KUKA KRL program: FrED_Main.src, FrED_Main.dat

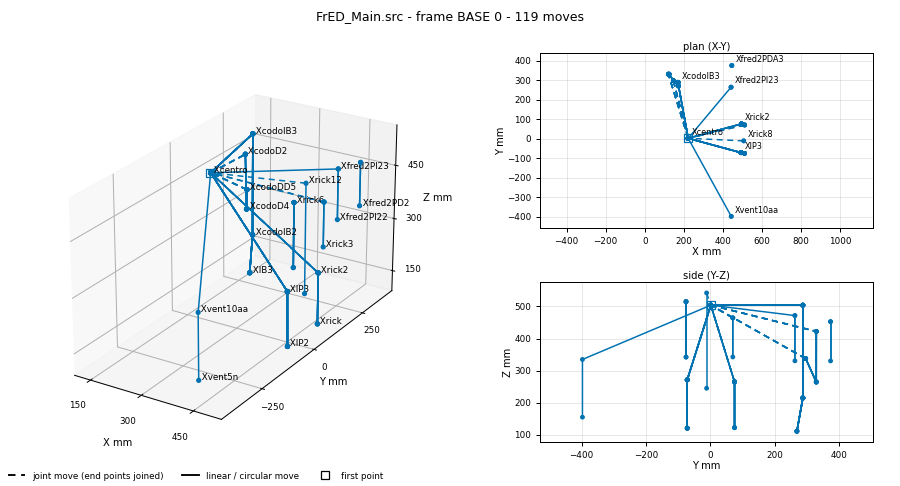
[picture p0: tool path of FrED_Main.src in frame BASE 0, 119 of 201 moves have a stored position in this frame; points joined in program order, loops and branches not executed]
--- FrED_Main.src ---
&ACCESS RVO
&PARAM DISKPATH = KRC:\R1\AAWS3
DEF codigoWS3( )
;FOLD INI;%{PE}
   DECL INT i
  ;FOLD BASISTECH INI
    GLOBAL INTERRUPT DECL 3 WHEN $STOPMESS==TRUE DO IR_STOPM ( )
    INTERRUPT ON 3
    BAS (#INITMOV,0 )

  ;ENDFOLD (BASISTECH INI)
;FOLD SPOTTECH INIw
USERSPOT(#INIT)
;ENDFOLD (SPOTTECH INI)
;FOLD GRIPPERTECH INI
USER_GRP(0,DUMMY,DUMMY,GDEFAULT)
;ENDFOLD (GRIPPERTECH INI)
;FOLD USER INI
  ;Make your modifications here
;ENDFOLD (USER INI)

;ENDFOLD (INI)

INTERRUPT DECL 25 WHEN NOT $IN[107] DO PAUSA()


;FOLD WAIT FOR ( IN 107 '' );%{PE}%R 8.3.40,%MKUKATPBASIS,%CEXT_WAIT_FOR,%VEXT_WAIT_FOR,%P 2:, 4:, 5:$IN, 6:107, 7:, 9:
WAIT FOR  ( $IN[107] )
;ENDFOLD
$OUT[105]=TRUE

INTERRUPT ON 25

FOR i= 1 to 2 STEP +1


;---------------------------------------------------------------------------------------------------------------------------------------------------------
;FRED 1


$OUT[101] = FALSE
WAIT SEC 0.5

;FOLD ; hola;%{PE}%R 8.3.40,%MKUKATPBASIS,%CCOMMENT,%VNORMAL,%P 2:hola
;ENDFOLD
;--- Movimiento a centro con velocidad reducida ---
PDAT_ACT=PPDAT4
FDAT_ACT=Fcentro
BAS(#PTP_PARAMS,20)
PTP Xcentro

;--- Abrir gripper ---
$OUT[101] = TRUE
$OUT[102] = FALSE
WAIT SEC 1

;--- Movimiento a codoIB3 ---
LDAT_ACT=LCPDAT2
FDAT_ACT=FcodoIB3
BAS(#CP_PARAMS,10)
LIN XcodoIB3

;--- Movimiento a codoIB2 ---
LDAT_ACT=LCPDAT5
FDAT_ACT=FcodoIB2
BAS(#CP_PARAMS,10)
LIN XcodoIB2

;FOLD LIN IB3 Vel=2 m/s CPDAT45 Tool[1]:navaja Base[0];%{PE}%R 8.3.40,%MKUKATPBASIS,%CMOVE,%VLIN,%P 1:LIN, 2:IB3, 3:, 5:2, 7:CPDAT45
$BWDSTART=FALSE
LDAT_ACT=LCPDAT45
FDAT_ACT=FIB3
BAS(#CP_PARAMS,2)
LIN XIB3
;ENDFOLD

;--- Cerrar gripper ---
$OUT[101] = FALSE
$OUT[102] = TRUE
WAIT SEC 1

;--- Regreso por codoIB2 ---
LDAT_ACT=LCPDAT5
FDAT_ACT=FcodoIB2
BAS(#CP_PARAMS,10)
LIN XcodoIB2

;--- Regreso por codoIB3 ---
LDAT_ACT=LCPDAT2
FDAT_ACT=FcodoIB3
BAS(#CP_PARAMS,10)
LIN XcodoIB3

;--- Regreso a centro ---
PDAT_ACT=PPDAT4
FDAT_ACT=Fcentro
BAS(#PTP_PARAMS,20)
PTP Xcentro

;FOLD LIN IP3 Vel=2 m/s CPDAT47 Tool[1]:navaja Base[0];%{PE}%R 8.3.40,%MKUKATPBASIS,%CMOVE,%VLIN,%P 1:LIN, 2:IP3, 3:, 5:2, 7:CPDAT47
$BWDSTART=FALSE
LDAT_ACT=LCPDAT47
FDAT_ACT=FIP3
BAS(#CP_PARAMS,2)
LIN XIP3
;ENDFOLD

;FOLD LIN IP2 Vel=2 m/s CPDAT46 Tool[1]:navaja Base[0];%{PE}%R 8.3.40,%MKUKATPBASIS,%CMOVE,%VLIN,%P 1:LIN, 2:IP2, 3:, 5:2, 7:CPDAT46
$BWDSTART=FALSE
LDAT_ACT=LCPDAT46
FDAT_ACT=FIP2
BAS(#CP_PARAMS,0.1)
LIN XIP2
;ENDFOLD


;--- Abrir gripper ---
$OUT[101] = TRUE
$OUT[102] = FALSE
WAIT SEC 1

;FOLD LIN IP4 Vel=2 m/s CPDAT47 Tool[1]:navaja Base[0];%{PE}%R 8.3.40,%MKUKATPBASIS,%CMOVE,%VLIN,%P 1:LIN, 2:IP4, 3:, 5:2, 7:CPDAT47
$BWDSTART=FALSE
LDAT_ACT=LCPDAT60
FDAT_ACT=FIP4
BAS(#CP_PARAMS,0.1)
LIN XIP4
;ENDFOLD



;--- Movimiento a centro ---
PDAT_ACT=PPDAT4
FDAT_ACT=Fcentro
BAS(#PTP_PARAMS,20)
PTP Xcentro

;--- Movimiento a codoD2 ---
PDAT_ACT=PPDAT6
FDAT_ACT=FcodoD2
BAS(#PTP_PARAMS,20)
PTP XcodoD2

;FOLD ; codoDnuevoagsrrar;%{PE}%R 8.3.40,%MKUKATPBASIS,%CCOMMENT,%VNORMAL,%P 2:codoDnuevoagsrrar
;ENDFOLD
;FOLD LIN codoD4 Vel=2 m/s CPDAT66 Tool[1]:navaja Base[0];%{PE}%R 8.3.40,%MKUKATPBASIS,%CMOVE,%VLIN,%P 1:LIN, 2:codoD4, 3:, 5:2, 7:CPDAT66
$BWDSTART=FALSE
LDAT_ACT=LCPDAT66
FDAT_ACT=FcodoD4
BAS(#CP_PARAMS,2)
LIN XcodoD4
;ENDFOLD

;--- Cerrar gripper ---
$OUT[101] = FALSE
$OUT[102] = TRUE
WAIT SEC 1

;FOLD LIN codoDD5 Vel=2 m/s CPDAT68 Tool[1]:navaja Base[0];%{PE}%R 8.3.40,%MKUKATPBASIS,%CMOVE,%VLIN,%P 1:LIN, 2:codoDD5, 3:, 5:2, 7:CPDAT68
$BWDSTART=FALSE
LDAT_ACT=LCPDAT68
FDAT_ACT=FcodoDD5
BAS(#CP_PARAMS,2)
LIN XcodoDD5
;ENDFOLD

;--- Movimiento a centro_5 con velocidad reducida ---
PDAT_ACT=PPDAT20
FDAT_ACT=Fcentro_5
BAS(#PTP_PARAMS,20)
PTP Xcentro_5

;FOLD LIN rick2 Vel=2 m/s CPDAT53 Tool[1]:navaja Base[0];%{PE}%R 8.3.40,%MKUKATPBASIS,%CMOVE,%VLIN,%P 1:LIN, 2:rick2, 3:, 5:2, 7:CPDAT53
$BWDSTART=FALSE
LDAT_ACT=LCPDAT53
FDAT_ACT=Frick2
BAS(#CP_PARAMS,2)
LIN Xrick2
;ENDFOLD

;FOLD LIN rick Vel=2 m/s CPDAT51 Tool[1]:navaja Base[0];%{PE}%R 8.3.40,%MKUKATPBASIS,%CMOVE,%VLIN,%P 1:LIN, 2:rick, 3:, 5:2, 7:CPDAT51
$BWDSTART=FALSE
LDAT_ACT=LCPDAT51
FDAT_ACT=Frick
BAS(#CP_PARAMS,0.1)
LIN Xrick
;ENDFOLD

;--- Abrir gripper ---
$OUT[101] = TRUE
$OUT[102] = FALSE
WAIT SEC 1

;FOLD LIN rick9 Vel=2 m/s CPDAT53 Tool[1]:navaja Base[0];%{PE}%R 8.3.40,%MKUKATPBASIS,%CMOVE,%VLIN,%P 1:LIN, 2:rick9, 3:, 5:2, 7:CPDAT53
$BWDSTART=FALSE
LDAT_ACT=LCPDAT61
FDAT_ACT=Frick9
BAS(#CP_PARAMS,0.1)
LIN Xrick9
;ENDFOLD

;--- Movimiento a centro ---
PDAT_ACT=PPDAT4
FDAT_ACT=Fcentro
BAS(#PTP_PARAMS,20)
PTP Xcentro

;FOLD LIN fred1PIA Vel=2 m/s CPDAT241 Tool[1]:navaja Base[0];%{PE}%R 8.3.40,%MKUKATPBASIS,%CMOVE,%VLIN,%P 1:LIN, 2:fred1PIA, 3:, 5:2, 7:CPDAT241
$BWDSTART=FALSE
LDAT_ACT=LCPDAT241
FDAT_ACT=Ffred1PIA
BAS(#CP_PARAMS,2)
LIN Xfred1PIA
;ENDFOLD

;FOLD LIN fred1PI Vel=2 m/s CPDAT240 Tool[1]:navaja Base[0];%{PE}%R 8.3.40,%MKUKATPBASIS,%CMOVE,%VLIN,%P 1:LIN, 2:fred1PI, 3:, 5:2, 7:CPDAT240
$BWDSTART=FALSE
LDAT_ACT=LCPDAT240
FDAT_ACT=Ffred1PI
BAS(#CP_PARAMS,2)
LIN Xfred1PI
;ENDFOLD

;--- Cerrar gripper ---
$OUT[101] = FALSE
$OUT[102] = TRUE
WAIT SEC 1

;FOLD LIN fred1PIA_1 Vel=2 m/s CPDAT241 Tool[1]:navaja Base[0];%{PE}%R 8.3.40,%MKUKATPBASIS,%CMOVE,%VLIN,%P 1:LIN, 2:fred1PIA_1, 3:, 5:2, 7:CPDAT241
$BWDSTART=FALSE
LDAT_ACT=LCPDAT244
FDAT_ACT=Ffred1PIA_1
BAS(#CP_PARAMS,2)
LIN Xfred1PIA_1
;ENDFOLD

;FOLD LIN rick6 Vel=2 m/s CPDAT57 Tool[1]:navaja Base[0];%{PE}%R 8.3.40,%MKUKATPBASIS,%CMOVE,%VLIN,%P 1:LIN, 2:rick6, 3:, 5:2, 7:CPDAT57
$BWDSTART=FALSE
LDAT_ACT=LCPDAT57
FDAT_ACT=Frick6
BAS(#CP_PARAMS,2)
LIN Xrick6
;ENDFOLD

;FOLD LIN rick5 Vel=2 m/s CPDAT56 Tool[1]:navaja Base[0];%{PE}%R 8.3.40,%MKUKATPBASIS,%CMOVE,%VLIN,%P 1:LIN, 2:rick5, 3:, 5:2, 7:CPDAT56
$BWDSTART=FALSE
LDAT_ACT=LCPDAT56
FDAT_ACT=Frick5
BAS(#CP_PARAMS,0.1)
LIN Xrick5
;ENDFOLD

;--- Abrir gripper ---
$OUT[101] = TRUE
$OUT[102] = FALSE
WAIT SEC 1

;FOLD LIN rick10 Vel=2 m/s CPDAT57 Tool[1]:navaja Base[0];%{PE}%R 8.3.40,%MKUKATPBASIS,%CMOVE,%VLIN,%P 1:LIN, 2:rick10, 3:, 5:2, 7:CPDAT57
$BWDSTART=FALSE
LDAT_ACT=LCPDAT62
FDAT_ACT=Frick10
BAS(#CP_PARAMS,1)
LIN Xrick10
;ENDFOLD


;FOLD ; perfil izq bueno arriba y luego abajo;%{PE}%R 8.3.40,%MKUKATPBASIS,%CCOMMENT,%VNORMAL,%P 2:perfil izq bueno arriba y luego abajo
;ENDFOLD

;FOLD LIN fred1PDA Vel=2 m/s CPDAT243 Tool[1]:navaja Base[0];%{PE}%R 8.3.40,%MKUKATPBASIS,%CMOVE,%VLIN,%P 1:LIN, 2:fred1PDA, 3:, 5:2, 7:CPDAT243
$BWDSTART=FALSE
LDAT_ACT=LCPDAT243
FDAT_ACT=Ffred1PDA
BAS(#CP_PARAMS,2)
LIN Xfred1PDA
;ENDFOLD


;FOLD LIN fred1PD Vel=2 m/s CPDAT242 Tool[1]:navaja Base[0];%{PE}%R 8.3.40,%MKUKATPBASIS,%CMOVE,%VLIN,%P 1:LIN, 2:fred1PD, 3:, 5:2, 7:CPDAT242
$BWDSTART=FALSE
LDAT_ACT=LCPDAT242
FDAT_ACT=Ffred1PD
BAS(#CP_PARAMS,2)
LIN Xfred1PD
;ENDFOLD

;--- Cerrar gripper ---
$OUT[101] = FALSE
$OUT[102] = TRUE
WAIT SEC 1

;FOLD LIN fred1PDA_1 Vel=2 m/s CPDAT243 Tool[1]:navaja Base[0];%{PE}%R 8.3.40,%MKUKATPBASIS,%CMOVE,%VLIN,%P 1:LIN, 2:fred1PDA_1, 3:, 5:2, 7:CPDAT243
$BWDSTART=FALSE
LDAT_ACT=LCPDAT245
FDAT_ACT=Ffred1PDA_1
BAS(#CP_PARAMS,2)
LIN Xfred1PDA_1
;ENDFOLD

;FOLD LIN rick4 Vel=2 m/s CPDAT55 Tool[1]:navaja Base[0];%{PE}%R 8.3.40,%MKUKATPBASIS,%CMOVE,%VLIN,%P 1:LIN, 2:rick4, 3:, 5:2, 7:CPDAT55
$BWDSTART=FALSE
LDAT_ACT=LCPDAT55
FDAT_ACT=Frick4
BAS(#CP_PARAMS,2)
LIN Xrick4
;ENDFOLD

;FOLD LIN rick3 Vel=2 m/s CPDAT54 Tool[1]:navaja Base[0];%{PE}%R 8.3.40,%MKUKATPBASIS,%CMOVE,%VLIN,%P 1:LIN, 2:rick3, 3:, 5:2, 7:CPDAT54
$BWDSTART=FALSE
LDAT_ACT=LCPDAT54
FDAT_ACT=Frick3
BAS(#CP_PARAMS,0.1)
LIN Xrick3
;ENDFOLD

;--- Abrir gripper ---
$OUT[101] = TRUE
$OUT[102] = FALSE
WAIT SEC 1

;FOLD LIN rick11 Vel=2 m/s CPDAT55 Tool[1]:navaja Base[0];%{PE}%R 8.3.40,%MKUKATPBASIS,%CMOVE,%VLIN,%P 1:LIN, 2:rick11, 3:, 5:2, 7:CPDAT55
$BWDSTART=FALSE
LDAT_ACT=LCPDAT63
FDAT_ACT=Frick11
BAS(#CP_PARAMS,1)
LIN Xrick11
;ENDFOLD

;--- Movimiento a centro ---
PDAT_ACT=PPDAT4
FDAT_ACT=Fcentro
BAS(#PTP_PARAMS,20)
PTP Xcentro

;FOLD LIN vent10aa Vel=2 m/s CPDAT70 Tool[1]:navaja Base[0];%{PE}%R 8.3.40,%MKUKATPBASIS,%CMOVE,%VLIN,%P 1:LIN, 2:vent10aa, 3:, 5:2, 7:CPDAT70
$BWDSTART=FALSE
LDAT_ACT=LCPDAT70
FDAT_ACT=Fvent10aa
BAS(#CP_PARAMS,2)
LIN Xvent10aa
;ENDFOLD

;FOLD LIN vent5n Vel=2 m/s CPDAT67 Tool[1]:navaja Base[0];%{PE}%R 8.3.40,%MKUKATPBASIS,%CMOVE,%VLIN,%P 1:LIN, 2:vent5n, 3:, 5:2, 7:CPDAT67
$BWDSTART=FALSE
LDAT_ACT=LCPDAT67
FDAT_ACT=Fvent5n
BAS(#CP_PARAMS,2)
LIN Xvent5n

;ENDFOLD
;--- Cerrar gripper ---
$OUT[101] = FALSE
$OUT[102] = TRUE
WAIT SEC 1

;FOLD LIN ventarribita Vel=2 m/s CPDAT247 Tool[1]:navaja Base[0];%{PE}%R 8.3.40,%MKUKATPBASIS,%CMOVE,%VLIN,%P 1:LIN, 2:ventarribita, 3:, 5:2, 7:CPDAT247
$BWDSTART=FALSE
LDAT_ACT=LCPDAT247
FDAT_ACT=Fventarribita
BAS(#CP_PARAMS,2)
LIN Xventarribita
;ENDFOLD

;--- Movimiento a vent88 ---
PDAT_ACT=PPDAT18
FDAT_ACT=Fvent88
BAS(#PTP_PARAMS,2)
PTP Xvent88

;FOLD LIN ventarriba Vel=2 m/s CPDAT239 Tool[1]:navaja Base[0];%{PE}%R 8.3.40,%MKUKATPBASIS,%CMOVE,%VLIN,%P 1:LIN, 2:ventarriba, 3:, 5:2, 7:CPDAT239
$BWDSTART=FALSE
LDAT_ACT=LCPDAT239
FDAT_ACT=Fventarriba
BAS(#CP_PARAMS,2)
LIN Xventarriba
;ENDFOLD

;FOLD LIN rick8 Vel=2 m/s CPDAT59 Tool[1]:navaja Base[0];%{PE}%R 8.3.40,%MKUKATPBASIS,%CMOVE,%VLIN,%P 1:LIN, 2:rick8, 3:, 5:2, 7:CPDAT59
$BWDSTART=FALSE
LDAT_ACT=LCPDAT59
FDAT_ACT=Frick8
BAS(#CP_PARAMS,.02)
LIN Xrick8
;ENDFOLD

;--- Abrir gripper ---
$OUT[101] = TRUE
$OUT[102] = FALSE
WAIT SEC 1

;FOLD LIN rick12 Vel=2 m/s CPDAT58 Tool[1]:navaja Base[0];%{PE}%R 8.3.40,%MKUKATPBASIS,%CMOVE,%VLIN,%P 1:LIN, 2:rick12, 3:, 5:2, 7:CPDAT58
$BWDSTART=FALSE
LDAT_ACT=LCPDAT64
FDAT_ACT=Frick12
BAS(#CP_PARAMS,2)
LIN Xrick12
;ENDFOLD

;--- Movimiento final a centro ---
PDAT_ACT=PPDAT4
FDAT_ACT=Fcentro
BAS(#PTP_PARAMS,20)
PTP Xcentro

;---------------------------------------------------------------------------------------------------------------------------------------------------------
;FRED 2
;---------------------------------------------------------------------------------------------------------------------------------------------------------

$OUT[101] = FALSE
WAIT SEC 0.5

;--- Movimiento a centro con velocidad reducida ---
PDAT_ACT=PPDAT4
FDAT_ACT=Fcentro
BAS(#PTP_PARAMS,20)
PTP Xcentro

;--- Abrir gripper ---
$OUT[101] = TRUE
$OUT[102] = FALSE
WAIT SEC 1

;--- Movimiento a codoIB3 ---
LDAT_ACT=LCPDAT2
FDAT_ACT=FcodoIB3
BAS(#CP_PARAMS,10)
LIN XcodoIB3

;--- Movimiento a codoIB2 ---
LDAT_ACT=LCPDAT5
FDAT_ACT=FcodoIB2
BAS(#CP_PARAMS,10)
LIN XcodoIB2

;FOLD LIN IB3 Vel=2 m/s CPDAT45 Tool[1]:navaja Base[0];%{PE}%R 8.3.40,%MKUKATPBASIS,%CMOVE,%VLIN,%P 1:LIN, 2:IB3, 3:, 5:2, 7:CPDAT45
$BWDSTART=FALSE
LDAT_ACT=LCPDAT45
FDAT_ACT=FIB3
BAS(#CP_PARAMS,2)
LIN XIB3
;ENDFOLD

;FOLD ; punto gripabajo IB3;%{PE}%R 8.3.40,%MKUKATPBASIS,%CCOMMENT,%VNORMAL,%P 2:punto gripabajo IB3
;ENDFOLD
;--- Cerrar gripper ---
$OUT[101] = FALSE
$OUT[102] = TRUE
WAIT SEC 1

;--- Regreso por codoIB2 ---
LDAT_ACT=LCPDAT5
FDAT_ACT=FcodoIB2
BAS(#CP_PARAMS,10)
LIN XcodoIB2

;--- Regreso por codoIB3 ---
LDAT_ACT=LCPDAT2
FDAT_ACT=FcodoIB3
BAS(#CP_PARAMS,10)
LIN XcodoIB3

;--- Regreso a centro ---
PDAT_ACT=PPDAT4
FDAT_ACT=Fcentro
BAS(#PTP_PARAMS,20)
PTP Xcentro


;FOLD LIN IP3 Vel=2 m/s CPDAT47 Tool[1]:navaja Base[0];%{PE}%R 8.3.40,%MKUKATPBASIS,%CMOVE,%VLIN,%P 1:LIN, 2:IP3, 3:, 5:2, 7:CPDAT47
$BWDSTART=FALSE
LDAT_ACT=LCPDAT47
FDAT_ACT=FIP3
BAS(#CP_PARAMS,2)
LIN XIP3
;ENDFOLD

;FOLD LIN IP2 Vel=2 m/s CPDAT46 Tool[1]:navaja Base[0];%{PE}%R 8.3.40,%MKUKATPBASIS,%CMOVE,%VLIN,%P 1:LIN, 2:IP2, 3:, 5:2, 7:CPDAT46
$BWDSTART=FALSE
LDAT_ACT=LCPDAT46
FDAT_ACT=FIP2
BAS(#CP_PARAMS,0.1)
LIN XIP2
;ENDFOLD

;--- Abrir gripper ---
$OUT[101] = TRUE
$OUT[102] = FALSE
WAIT SEC 1

;FOLD LIN IP4 Vel=2 m/s CPDAT47 Tool[1]:navaja Base[0];%{PE}%R 8.3.40,%MKUKATPBASIS,%CMOVE,%VLIN,%P 1:LIN, 2:IP4, 3:, 5:2, 7:CPDAT47
$BWDSTART=FALSE
LDAT_ACT=LCPDAT60
FDAT_ACT=FIP4
BAS(#CP_PARAMS,0.1)
LIN XIP4
;ENDFOLD


;--- Movimiento a centro ---
PDAT_ACT=PPDAT4
FDAT_ACT=Fcentro
BAS(#PTP_PARAMS,20)
PTP Xcentro

;--- Movimiento a codoD2 ---
PDAT_ACT=PPDAT6
FDAT_ACT=FcodoD2
BAS(#PTP_PARAMS,20)
PTP XcodoD2


;FOLD LIN codoD4 Vel=2 m/s CPDAT66 Tool[1]:navaja Base[0];%{PE}%R 8.3.40,%MKUKATPBASIS,%CMOVE,%VLIN,%P 1:LIN, 2:codoD4, 3:, 5:2, 7:CPDAT66
$BWDSTART=FALSE
LDAT_ACT=LCPDAT66
FDAT_ACT=FcodoD4
BAS(#CP_PARAMS,2)
LIN XcodoD4
;ENDFOLD

;--- Cerrar gripper ---
$OUT[101] = FALSE
$OUT[102] = TRUE
WAIT SEC 1

;FOLD LIN codoDD5 Vel=2 m/s CPDAT68 Tool[1]:navaja Base[0];%{PE}%R 8.3.40,%MKUKATPBASIS,%CMOVE,%VLIN,%P 1:LIN, 2:codoDD5, 3:, 5:2, 7:CPDAT68
$BWDSTART=FALSE
LDAT_ACT=LCPDAT68
FDAT_ACT=FcodoDD5
BAS(#CP_PARAMS,2)
LIN XcodoDD5
;ENDFOLD

;--- Movimiento a centro_5 con velocidad reducida ---
PDAT_ACT=PPDAT20
FDAT_ACT=Fcentro_5
BAS(#PTP_PARAMS,20)
PTP Xcentro_5

;FOLD LIN rick2 Vel=2 m/s CPDAT53 Tool[1]:navaja Base[0];%{PE}%R 8.3.40,%MKUKATPBASIS,%CMOVE,%VLIN,%P 1:LIN, 2:rick2, 3:, 5:2, 7:CPDAT53
$BWDSTART=FALSE
LDAT_ACT=LCPDAT53
FDAT_ACT=Frick2
BAS(#CP_PARAMS,2)
LIN Xrick2
;ENDFOLD

;FOLD LIN rick Vel=2 m/s CPDAT51 Tool[1]:navaja Base[0];%{PE}%R 8.3.40,%MKUKATPBASIS,%CMOVE,%VLIN,%P 1:LIN, 2:rick, 3:, 5:2, 7:CPDAT51
$BWDSTART=FALSE
LDAT_ACT=LCPDAT51
FDAT_ACT=Frick
BAS(#CP_PARAMS,0.1)
LIN Xrick
;ENDFOLD

;--- Abrir gripper ---
$OUT[101] = TRUE
$OUT[102] = FALSE
WAIT SEC 1

;FOLD LIN rick9 Vel=2 m/s CPDAT53 Tool[1]:navaja Base[0];%{PE}%R 8.3.40,%MKUKATPBASIS,%CMOVE,%VLIN,%P 1:LIN, 2:rick9, 3:, 5:2, 7:CPDAT53
$BWDSTART=FALSE
LDAT_ACT=LCPDAT61
FDAT_ACT=Frick9
BAS(#CP_PARAMS,0.1)
LIN Xrick9
;ENDFOLD

;--- Movimiento a centro ---
PDAT_ACT=PPDAT4
FDAT_ACT=Fcentro
BAS(#PTP_PARAMS,20)
PTP Xcentro

;PERFIL IZQUIERDO2 ARRIBA
$BWDSTART=FALSE
LDAT_ACT=LCPDAT101
FDAT_ACT=Ffred2PI23
BAS(#CP_PARAMS,2)
LIN Xfred2PI23

;PERFIL IZQUIERDO2 ABAJO
$BWDSTART=FALSE
LDAT_ACT=LCPDAT100
FDAT_ACT=Ffred2PI22
BAS(#CP_PARAMS,2)
LIN Xfred2PI22

;--- Cerrar gripper ---
$OUT[101] = FALSE
$OUT[102] = TRUE
WAIT SEC 1

;PERFIL IZQUIERDO2 ARRIBA
$BWDSTART=FALSE
LDAT_ACT=LCPDAT102
FDAT_ACT=Ffred2PI24
BAS(#CP_PARAMS,2)
LIN Xfred2PI24


;este se borra creo
;$BWDSTART=FALSE
;LDAT_ACT=LCPDAT260
;FDAT_ACT=Frick68
;BAS(#CP_PARAMS,2)
;LIN Xrick68


;FOLD LIN fred2PIA Vel=2 m/s CPDAT264 Tool[1]:navaja Base[0];%{PE}%R 8.3.40,%MKUKATPBASIS,%CMOVE,%VLIN,%P 1:LIN, 2:fred2PIA, 3:, 5:2, 7:CPDAT264
$BWDSTART=FALSE
LDAT_ACT=LCPDAT264
FDAT_ACT=Ffred2PIA
BAS(#CP_PARAMS,2)
LIN Xfred2PIA
;ENDFOLD

;FOLD LIN fred2PII Vel=2 m/s CPDAT263 Tool[1]:navaja Base[0];%{PE}%R 8.3.40,%MKUKATPBASIS,%CMOVE,%VLIN,%P 1:LIN, 2:fred2PII, 3:, 5:2, 7:CPDAT263
$BWDSTART=FALSE
LDAT_ACT=LCPDAT263
FDAT_ACT=Ffred2PII
BAS(#CP_PARAMS,0.1)
LIN Xfred2PII
;ENDFOLD

;este se borra creo
;$BWDSTART=FALSE
;LDAT_ACT=LCPDAT261
;FDAT_ACT=Frick69
;BAS(#CP_PARAMS,2)
;LIN Xrick69

;--- Abrir gripper ---
$OUT[101] = TRUE
$OUT[102] = FALSE
WAIT SEC 1

;FOLD LIN fred2PIAA Vel=2 m/s CPDAT265 Tool[1]:navaja Base[0];%{PE}%R 8.3.40,%MKUKATPBASIS,%CMOVE,%VLIN,%P 1:LIN, 2:fred2PIAA, 3:, 5:2, 7:CPDAT265
$BWDSTART=FALSE
LDAT_ACT=LCPDAT265
FDAT_ACT=Ffred2PIAA
BAS(#CP_PARAMS,0.1)
LIN Xfred2PIAA
;ENDFOLD

;este se borra creo
;$BWDSTART=FALSE
;LDAT_ACT=LCPDAT262
;FDAT_ACT=Frick70
;BAS(#CP_PARAMS,2)
;LIN Xrick70


;PERFILDERECHO2 ARRIBA
$BWDSTART=FALSE
LDAT_ACT=LCPDAT104
FDAT_ACT=Ffred2PDA3
BAS(#CP_PARAMS,2)
LIN Xfred2PDA3


;PERFILDERECHO2 ABAJO
$BWDSTART=FALSE
LDAT_ACT=LCPDAT103
FDAT_ACT=Ffred2PD2
BAS(#CP_PARAMS,2)
LIN Xfred2PD2

;--- Cerrar gripper ---
$OUT[101] = FALSE
$OUT[102] = TRUE
WAIT SEC 1

;PERFILDERECHO2 ARRIBA
$BWDSTART=FALSE
LDAT_ACT=LCPDAT105
FDAT_ACT=Ffred2PDA4
BAS(#CP_PARAMS,2)
LIN Xfred2PDA4

;FOLD LIN fred2pdpa Vel=2 m/s CPDAT259 Tool[1]:navaja Base[0];%{PE}%R 8.3.40,%MKUKATPBASIS,%CMOVE,%VLIN,%P 1:LIN, 2:fred2pdpa, 3:, 5:2, 7:CPDAT259
$BWDSTART=FALSE
LDAT_ACT=LCPDAT259
FDAT_ACT=Ffred2pdpa
BAS(#CP_PARAMS,2)
LIN Xfred2pdpa
;ENDFOLD

;FOLD LIN fred2PDP Vel=2 m/s CPDAT257 Tool[1]:navaja Base[0];%{PE}%R 8.3.40,%MKUKATPBASIS,%CMOVE,%VLIN,%P 1:LIN, 2:fred2PDP, 3:, 5:2, 7:CPDAT257
$BWDSTART=FALSE
LDAT_ACT=LCPDAT257
FDAT_ACT=Ffred2PDP
BAS(#CP_PARAMS,0.1)
LIN Xfred2PDP
;ENDFOLD

;--- Abrir gripper ---
$OUT[101] = TRUE
$OUT[102] = FALSE
WAIT SEC 1

;FOLD LIN fred3pdpa Vel=2 m/s CPDAT258 Tool[1]:navaja Base[0];%{PE}%R 8.3.40,%MKUKATPBASIS,%CMOVE,%VLIN,%P 1:LIN, 2:fred3pdpa, 3:, 5:2, 7:CPDAT258
$BWDSTART=FALSE
LDAT_ACT=LCPDAT258
FDAT_ACT=Ffred3pdpa
BAS(#CP_PARAMS,0.1)
LIN Xfred3pdpa
;ENDFOLD

;--- Movimiento a centro ---
PDAT_ACT=PPDAT4
FDAT_ACT=Fcentro
BAS(#PTP_PARAMS,20)
PTP Xcentro

;FOLD LIN ventfred2ARRIBA Vel=2 m/s CPDAT250 Tool[1]:navaja Base[0];%{PE}%R 8.3.40,%MKUKATPBASIS,%CMOVE,%VLIN,%P 1:LIN, 2:ventfred2ARRIBA, 3:, 5:2, 7:CPDAT250
$BWDSTART=FALSE
LDAT_ACT=LCPDAT250
FDAT_ACT=Fventfred2ARRIBA
BAS(#CP_PARAMS,2)
LIN Xventfred2ARRIBA
;ENDFOLD



;FOLD LIN ventfred2 Vel=2 m/s CPDAT249 Tool[1]:navaja Base[0];%{PE}%R 8.3.40,%MKUKATPBASIS,%CMOVE,%VLIN,%P 1:LIN, 2:ventfred2, 3:, 5:2, 7:CPDAT249
$BWDSTART=FALSE
LDAT_ACT=LCPDAT249
FDAT_ACT=Fventfred2
BAS(#CP_PARAMS,2)
LIN Xventfred2
;ENDFOLD

;--- Cerrar gripper ---
$OUT[101] = FALSE
$OUT[102] = TRUE
WAIT SEC 1

;FOLD LIN ventfred2ARRIBA Vel=2 m/s CPDAT250 Tool[1]:navaja Base[0];%{PE}%R 8.3.40,%MKUKATPBASIS,%CMOVE,%VLIN,%P 1:LIN, 2:ventfred2ARRIBA, 3:, 5:2, 7:CPDAT250
$BWDSTART=FALSE
LDAT_ACT=LCPDAT250
FDAT_ACT=Fventfred2ARRIBA
BAS(#CP_PARAMS,2)
LIN Xventfred2ARRIBA
;ENDFOLD

;--- Movimiento a vent88 ---
PDAT_ACT=PPDAT18
FDAT_ACT=Fvent88
BAS(#PTP_PARAMS,2)
PTP Xvent88


;FOLD LIN ventarriba_1 Vel=2 m/s CPDAT239 Tool[1]:navaja Base[0];%{PE}%R 8.3.40,%MKUKATPBASIS,%CMOVE,%VLIN,%P 1:LIN, 2:ventarriba_1, 3:, 5:2, 7:CPDAT239
$BWDSTART=FALSE
LDAT_ACT=LCPDAT288
FDAT_ACT=Fventarriba_1
BAS(#CP_PARAMS,2)
LIN Xventarriba_1
;ENDFOLD

;FOLD LIN rick71 Vel=2 m/s CPDAT59 Tool[1]:navaja Base[0];%{PE}%R 8.3.40,%MKUKATPBASIS,%CMOVE,%VLIN,%P 1:LIN, 2:rick71, 3:, 5:2, 7:CPDAT59
$BWDSTART=FALSE
LDAT_ACT=LCPDAT289
FDAT_ACT=Frick71
BAS(#CP_PARAMS,0.02)
LIN Xrick71
;ENDFOLD

;--- Abrir gripper ---
$OUT[101] = TRUE
$OUT[102] = FALSE
WAIT SEC 1

;FOLD LIN rick72 Vel=2 m/s CPDAT58 Tool[1]:navaja Base[0];%{PE}%R 8.3.40,%MKUKATPBASIS,%CMOVE,%VLIN,%P 1:LIN, 2:rick72, 3:, 5:2, 7:CPDAT58
$BWDSTART=FALSE
LDAT_ACT=LCPDAT290
FDAT_ACT=Frick72
BAS(#CP_PARAMS,2)
LIN Xrick72
;ENDFOLD


;--- Movimiento final a centro ---
PDAT_ACT=PPDAT4
FDAT_ACT=Fcentro
BAS(#PTP_PARAMS,20)
PTP Xcentro


;---------------------------------------------------------------------------------------------------------------------------------------------------------
;FRED 3;---------------------------------------------------------------------------------------------------------------------------------------------------------

$OUT[101] = FALSE
WAIT SEC 0.5

;--- Movimiento a centro con velocidad reducida ---
PDAT_ACT=PPDAT4
FDAT_ACT=Fcentro
BAS(#PTP_PARAMS,20)
PTP Xcentro

;--- Abrir gripper ---
$OUT[101] = TRUE
$OUT[102] = FALSE
WAIT SEC 1

;--- Movimiento a codoIB3 ---
LDAT_ACT=LCPDAT2
FDAT_ACT=FcodoIB3
BAS(#CP_PARAMS,10)
LIN XcodoIB3

;--- Movimiento a codoIB2 ---
LDAT_ACT=LCPDAT5
FDAT_ACT=FcodoIB2
BAS(#CP_PARAMS,10)
LIN XcodoIB2

;FOLD LIN IB3 Vel=2 m/s CPDAT45 Tool[1]:navaja Base[0];%{PE}%R 8.3.40,%MKUKATPBASIS,%CMOVE,%VLIN,%P 1:LIN, 2:IB3, 3:, 5:2, 7:CPDAT45
$BWDSTART=FALSE
LDAT_ACT=LCPDAT45
FDAT_ACT=FIB3
BAS(#CP_PARAMS,2)
LIN XIB3
;ENDFOLD

;--- Cerrar gripper ---
$OUT[101] = FALSE
$OUT[102] = TRUE
WAIT SEC 1

;--- Regreso por codoIB2 ---
LDAT_ACT=LCPDAT5
FDAT_ACT=FcodoIB2
BAS(#CP_PARAMS,10)
LIN XcodoIB2

;--- Regreso por codoIB3 ---
LDAT_ACT=LCPDAT2
FDAT_ACT=FcodoIB3
BAS(#CP_PARAMS,10)
LIN XcodoIB3

;--- Regreso a centro ---
PDAT_ACT=PPDAT4
FDAT_ACT=Fcentro
BAS(#PTP_PARAMS,20)
PTP Xcentro

;FOLD LIN IP3 Vel=2 m/s CPDAT47 Tool[1]:navaja Base[0];%{PE}%R 8.3.40,%MKUKATPBASIS,%CMOVE,%VLIN,%P 1:LIN, 2:IP3, 3:, 5:2, 7:CPDAT47
$BWDSTART=FALSE
LDAT_ACT=LCPDAT47
FDAT_ACT=FIP3
BAS(#CP_PARAMS,2)
LIN XIP3
;ENDFOLD

;FOLD LIN IP2 Vel=2 m/s CPDAT46 Tool[1]:navaja Base[0];%{PE}%R 8.3.40,%MKUKATPBASIS,%CMOVE,%VLIN,%P 1:LIN, 2:IP2, 3:, 5:2, 7:CPDAT46
$BWDSTART=FALSE
LDAT_ACT=LCPDAT46
FDAT_ACT=FIP2
BAS(#CP_PARAMS,0.1)
LIN XIP2
;ENDFOLD

;--- Abrir gripper ---
$OUT[101] = TRUE
$OUT[102] = FALSE
WAIT SEC 1

;FOLD LIN IP4 Vel=2 m/s CPDAT47 Tool[1]:navaja Base[0];%{PE}%R 8.3.40,%MKUKATPBASIS,%CMOVE,%VLIN,%P 1:LIN, 2:IP4, 3:, 5:2, 7:CPDAT47
$BWDSTART=FALSE
LDAT_ACT=LCPDAT60
FDAT_ACT=FIP4
BAS(#CP_PARAMS,0.1)
LIN XIP4
;ENDFOLD


;--- Movimiento a centro ---
PDAT_ACT=PPDAT4
FDAT_ACT=Fcentro
BAS(#PTP_PARAMS,20)
PTP Xcentro

;--- Movimiento a codoD2 ---
PDAT_ACT=PPDAT6
FDAT_ACT=FcodoD2
BAS(#PTP_PARAMS,20)
PTP XcodoD2



;FOLD ; codoDnuevoagsrrar;%{PE}%R 8.3.40,%MKUKATPBASIS,%CCOMMENT,%VNORMAL,%P 2:codoDnuevoagsrrar
;ENDFOLD

;FOLD LIN codoD4 Vel=2 m/s CPDAT66 Tool[1]:navaja Base[0];%{PE}%R 8.3.40,%MKUKATPBASIS,%CMOVE,%VLIN,%P 1:LIN, 2:codoD4, 3:, 5:2, 7:CPDAT66
$BWDSTART=FALSE
LDAT_ACT=LCPDAT66
FDAT_ACT=FcodoD4
BAS(#CP_PARAMS,2)
LIN XcodoD4
;ENDFOLD

;--- Cerrar gripper ---
$OUT[101] = FALSE
$OUT[102] = TRUE
WAIT SEC 1

;FOLD LIN codoDD5 Vel=2 m/s CPDAT68 Tool[1]:navaja Base[0];%{PE}%R 8.3.40,%MKUKATPBASIS,%CMOVE,%VLIN,%P 1:LIN, 2:codoDD5, 3:, 5:2, 7:CPDAT68
$BWDSTART=FALSE
LDAT_ACT=LCPDAT68
FDAT_ACT=FcodoDD5
BAS(#CP_PARAMS,2)
LIN XcodoDD5
;ENDFOLD

;--- Movimiento a centro_5 con velocidad reducida ---
PDAT_ACT=PPDAT20
FDAT_ACT=Fcentro_5
BAS(#PTP_PARAMS,20)
PTP Xcentro_5

;FOLD LIN rick2 Vel=2 m/s CPDAT53 Tool[1]:navaja Base[0];%{PE}%R 8.3.40,%MKUKATPBASIS,%CMOVE,%VLIN,%P 1:LIN, 2:rick2, 3:, 5:2, 7:CPDAT53
$BWDSTART=FALSE
LDAT_ACT=LCPDAT53
FDAT_ACT=Frick2
BAS(#CP_PARAMS,2)
LIN Xrick2
;ENDFOLD

;FOLD LIN rick Vel=2 m/s CPDAT51 Tool[1]:navaja Base[0];%{PE}%R 8.3.40,%MKUKATPBASIS,%CMOVE,%VLIN,%P 1:LIN, 2:rick, 3:, 5:2, 7:CPDAT51
$BWDSTART=FALSE
LDAT_ACT=LCPDAT51
FDAT_ACT=Frick
BAS(#CP_PARAMS,0.1)
LIN Xrick
;ENDFOLD

;--- Abrir gripper ---
$OUT[101] = TRUE
$OUT[102] = FALSE
WAIT SEC 1

;FOLD LIN rick9 Vel=2 m/s CPDAT53 Tool[1]:navaja Base[0];%{PE}%R 8.3.40,%MKUKATPBASIS,%CMOVE,%VLIN,%P 1:LIN, 2:rick9, 3:, 5:2, 7:CPDAT53
$BWDSTART=FALSE
LDAT_ACT=LCPDAT61
FDAT_ACT=Frick9
BAS(#CP_PARAMS,0.1)
LIN Xrick9
;ENDFOLD

;--- Movimiento a centro ---
PDAT_ACT=PPDAT4
FDAT_ACT=Fcentro
BAS(#PTP_PARAMS,20)
PTP Xcentro

;PERFILIZQUEIRDO3 ARRIBA
$BWDSTART=FALSE
LDAT_ACT=LCPDAT167
FDAT_ACT=Ffred3PIA
BAS(#CP_PARAMS,2)
LIN Xfred3PIA


;PERFILIZQUIERDO3 ABAJO
$BWDSTART=FALSE
LDAT_ACT=LCPDAT166
FDAT_ACT=FfreD3PI
BAS(#CP_PARAMS,2)
LIN XfreD3PI

;--- Cerrar gripper ---
$OUT[101] = FALSE
$OUT[102] = TRUE
WAIT SEC 1

;PERFILIZQUIERDO3 ARRIBA
$BWDSTART=FALSE
LDAT_ACT=LCPDAT170
FDAT_ACT=Ffred3PIA_1
BAS(#CP_PARAMS,2)
LIN Xfred3PIA_1

;FOLD LIN rick6 Vel=2 m/s CPDAT57 Tool[1]:navaja Base[0];%{PE}%R 8.3.40,%MKUKATPBASIS,%CMOVE,%VLIN,%P 1:LIN, 2:rick6, 3:, 5:2, 7:CPDAT57
$BWDSTART=FALSE
LDAT_ACT=LCPDAT57
FDAT_ACT=Frick6
BAS(#CP_PARAMS,2)
LIN Xrick6
;ENDFOLD

;FOLD LIN rick5 Vel=2 m/s CPDAT56 Tool[1]:navaja Base[0];%{PE}%R 8.3.40,%MKUKATPBASIS,%CMOVE,%VLIN,%P 1:LIN, 2:rick5, 3:, 5:2, 7:CPDAT56
$BWDSTART=FALSE
LDAT_ACT=LCPDAT56
FDAT_ACT=Frick5
BAS(#CP_PARAMS,0.1)
LIN Xrick5
;ENDFOLD

;--- Abrir gripper ---
$OUT[101] = TRUE
$OUT[102] = FALSE
WAIT SEC 1

;FOLD LIN rick10 Vel=2 m/s CPDAT57 Tool[1]:navaja Base[0];%{PE}%R 8.3.40,%MKUKATPBASIS,%CMOVE,%VLIN,%P 1:LIN, 2:rick10, 3:, 5:2, 7:CPDAT57
$BWDSTART=FALSE
LDAT_ACT=LCPDAT62
FDAT_ACT=Frick10
BAS(#CP_PARAMS,0.1)
LIN Xrick10
;ENDFOLD


;FOLD ; perfil izq bueno arriba y luego abajo;%{PE}%R 8.3.40,%MKUKATPBASIS,%CCOMMENT,%VNORMAL,%P 2:perfil izq bueno arriba y luego abajo
;ENDFOLD

;PERFILDERECHO3 ARRIBA
$BWDSTART=FALSE
LDAT_ACT=LCPDAT169
FDAT_ACT=Ffred3PD4
BAS(#CP_PARAMS,2)
LIN Xfred3PD4


;PERFILDERECHO3 ABAJO
$BWDSTART=FALSE
LDAT_ACT=LCPDAT168
FDAT_ACT=Ffred3PD3
BAS(#CP_PARAMS,2)
LIN Xfred3PD3

;--- Cerrar gripper ---
$OUT[101] = FALSE
$OUT[102] = TRUE
WAIT SEC 1

;PERFILDERECHO3 ARRIBA
$BWDSTART=FALSE
LDAT_ACT=LCPDAT171
FDAT_ACT=Ffred3PD5
BAS(#CP_PARAMS,2)
LIN Xfred3PD5

;FOLD LIN fred33PDA Vel=2 m/s CPDAT55 Tool[1]:navaja Base[0];%{PE}%R 8.3.40,%MKUKATPBASIS,%CMOVE,%VLIN,%P 1:LIN, 2:fred33PDA, 3:, 5:2, 7:CPDAT55
$BWDSTART=FALSE
LDAT_ACT=LCPDAT55
FDAT_ACT=Ffred33PDA
BAS(#CP_PARAMS,2)
LIN Xfred33PDA
;ENDFOLD

;FOLD LIN fred3PDD Vel=2 m/s CPDAT54 Tool[1]:navaja Base[0];%{PE}%R 8.3.40,%MKUKATPBASIS,%CMOVE,%VLIN,%P 1:LIN, 2:fred3PDD, 3:, 5:2, 7:CPDAT54
$BWDSTART=FALSE
LDAT_ACT=LCPDAT54
FDAT_ACT=Ffred3PDD
BAS(#CP_PARAMS,0.1)
LIN Xfred3PDD
;ENDFOLD

;--- Abrir gripper ---
$OUT[101] = TRUE
$OUT[102] = FALSE
WAIT SEC 1

;FOLD LIN rick11 Vel=2 m/s CPDAT55 Tool[1]:navaja Base[0];%{PE}%R 8.3.40,%MKUKATPBASIS,%CMOVE,%VLIN,%P 1:LIN, 2:rick11, 3:, 5:2, 7:CPDAT55
$BWDSTART=FALSE
LDAT_ACT=LCPDAT63
FDAT_ACT=Frick11
BAS(#CP_PARAMS,0.1)
LIN Xrick11
;ENDFOLD

;--- Movimiento a centro ---
PDAT_ACT=PPDAT4
FDAT_ACT=Fcentro
BAS(#PTP_PARAMS,20)
PTP Xcentro

;FOLD LIN ventfred3ARRIBA Vel=2 m/s CPDAT252 Tool[1]:navaja Base[0];%{PE}%R 8.3.40,%MKUKATPBASIS,%CMOVE,%VLIN,%P 1:LIN, 2:ventfred3ARRIBA, 3:, 5:2, 7:CPDAT252
$BWDSTART=FALSE
LDAT_ACT=LCPDAT252
FDAT_ACT=Fventfred3ARRIBA
BAS(#CP_PARAMS,2)
LIN Xventfred3ARRIBA
;ENDFOLD

;FOLD LIN ventfred3 Vel=2 m/s CPDAT251 Tool[1]:navaja Base[0];%{PE}%R 8.3.40,%MKUKATPBASIS,%CMOVE,%VLIN,%P 1:LIN, 2:ventfred3, 3:, 5:2, 7:CPDAT251
$BWDSTART=FALSE
LDAT_ACT=LCPDAT251
FDAT_ACT=Fventfred3
BAS(#CP_PARAMS,2)
LIN Xventfred3
;ENDFOLD


;--- Cerrar gripper ---
$OUT[101] = FALSE
$OUT[102] = TRUE
WAIT SEC 1


$BWDSTART=FALSE
LDAT_ACT=LCPDAT252
FDAT_ACT=Fventfred3ARRIBA
BAS(#CP_PARAMS,2)
LIN Xventfred3ARRIBA


;--- Movimiento a vent88 ---
PDAT_ACT=PPDAT18
FDAT_ACT=Fvent88
BAS(#PTP_PARAMS,2)
PTP Xvent88

;FOLD LIN ventarriba_2 Vel=2 m/s CPDAT239 Tool[1]:navaja Base[0];%{PE}%R 8.3.40,%MKUKATPBASIS,%CMOVE,%VLIN,%P 1:LIN, 2:ventarriba_2, 3:, 5:2, 7:CPDAT239
$BWDSTART=FALSE
LDAT_ACT=LCPDAT291
FDAT_ACT=Fventarriba_2
BAS(#CP_PARAMS,2)
LIN Xventarriba_2
;ENDFOLD

;FOLD LIN rick73 Vel=2 m/s CPDAT59 Tool[1]:navaja Base[0];%{PE}%R 8.3.40,%MKUKATPBASIS,%CMOVE,%VLIN,%P 1:LIN, 2:rick73, 3:, 5:2, 7:CPDAT59
$BWDSTART=FALSE
LDAT_ACT=LCPDAT292
FDAT_ACT=Frick73
BAS(#CP_PARAMS,0.02)
LIN Xrick73
;ENDFOLD

;--- Abrir gripper ---
$OUT[101] = TRUE
$OUT[102] = FALSE
WAIT SEC 1

;FOLD LIN rick74 Vel=2 m/s CPDAT58 Tool[1]:navaja Base[0];%{PE}%R 8.3.40,%MKUKATPBASIS,%CMOVE,%VLIN,%P 1:LIN, 2:rick74, 3:, 5:2, 7:CPDAT58
$BWDSTART=FALSE
LDAT_ACT=LCPDAT293
FDAT_ACT=Frick74
BAS(#CP_PARAMS,2)
LIN Xrick74
;ENDFOLD



;--- Movimiento final a centro ---
PDAT_ACT=PPDAT4
FDAT_ACT=Fcentro
BAS(#PTP_PARAMS,20)
PTP Xcentro

;---------------------------------------------------------------------------------------------------------------------------------------------------------
;FRED 4;---------------------------------------------------------------------------------------------------------------------------------------------------------

$OUT[101] = FALSE
WAIT SEC 0.5

;--- Movimiento a centro con velocidad reducida ---
PDAT_ACT=PPDAT4
FDAT_ACT=Fcentro
BAS(#PTP_PARAMS,20)
PTP Xcentro

;--- Abrir gripper ---
$OUT[101] = TRUE
$OUT[102] = FALSE
WAIT SEC 1

;--- Movimiento a codoIB3 ---
LDAT_ACT=LCPDAT2
FDAT_ACT=FcodoIB3
BAS(#CP_PARAMS,10)
LIN XcodoIB3

;--- Movimiento a codoIB2 ---
LDAT_ACT=LCPDAT5
FDAT_ACT=FcodoIB2
BAS(#CP_PARAMS,10)
LIN XcodoIB2


$BWDSTART=FALSE
LDAT_ACT=LCPDAT45
FDAT_ACT=FIB3
BAS(#CP_PARAMS,2)
LIN XIB3

;--- Cerrar gripper ---
$OUT[101] = FALSE
$OUT[102] = TRUE
WAIT SEC 1

;--- Regreso por codoIB2 ---
LDAT_ACT=LCPDAT5
FDAT_ACT=FcodoIB2
BAS(#CP_PARAMS,10)
LIN XcodoIB2

;--- Regreso por codoIB3 ---
LDAT_ACT=LCPDAT2
FDAT_ACT=FcodoIB3
BAS(#CP_PARAMS,10)
LIN XcodoIB3

;--- Regreso a centro ---
PDAT_ACT=PPDAT4
FDAT_ACT=Fcentro
BAS(#PTP_PARAMS,20)
PTP Xcentro


$BWDSTART=FALSE
LDAT_ACT=LCPDAT47
FDAT_ACT=FIP3
BAS(#CP_PARAMS,2)
LIN XIP3



$BWDSTART=FALSE
LDAT_ACT=LCPDAT46
FDAT_ACT=FIP2
BAS(#CP_PARAMS,0.1)
LIN XIP2


;--- Abrir gripper ---
$OUT[101] = TRUE
$OUT[102] = FALSE
WAIT SEC 1


$BWDSTART=FALSE
LDAT_ACT=LCPDAT60
FDAT_ACT=FIP4
BAS(#CP_PARAMS,0.1)
LIN XIP4
;


;--- Movimiento a centro ---
PDAT_ACT=PPDAT4
FDAT_ACT=Fcentro
BAS(#PTP_PARAMS,20)
PTP Xcentro

;--- Movimiento a codoD2 ---
PDAT_ACT=PPDAT6
FDAT_ACT=FcodoD2
BAS(#PTP_PARAMS,20)
PTP XcodoD2

$BWDSTART=FALSE
LDAT_ACT=LCPDAT66
FDAT_ACT=FcodoD4
BAS(#CP_PARAMS,2)
LIN XcodoD4


;--- Cerrar gripper ---
$OUT[101] = FALSE
$OUT[102] = TRUE
WAIT SEC 1

$BWDSTART=FALSE
LDAT_ACT=LCPDAT68
FDAT_ACT=FcodoDD5
BAS(#CP_PARAMS,2)
LIN XcodoDD5


;--- Movimiento a centro_5 con velocidad reducida ---
PDAT_ACT=PPDAT20
FDAT_ACT=Fcentro_5
BAS(#PTP_PARAMS,20)
PTP Xcentro_5




;FOLD LIN fred5codoDA Vel=2 m/s CPDAT305 Tool[1]:navaja Base[0];%{PE}%R 8.3.40,%MKUKATPBASIS,%CMOVE,%VLIN,%P 1:LIN, 2:fred5codoDA, 3:, 5:2, 7:CPDAT305
$BWDSTART=FALSE
LDAT_ACT=LCPDAT305
FDAT_ACT=Ffred5codoDA
BAS(#CP_PARAMS,2)
LIN Xfred5codoDA
;ENDFOLD

;FOLD LIN fred5codoD Vel=2 m/s CPDAT304 Tool[1]:navaja Base[0];%{PE}%R 8.3.40,%MKUKATPBASIS,%CMOVE,%VLIN,%P 1:LIN, 2:fred5codoD, 3:, 5:2, 7:CPDAT304
$BWDSTART=FALSE
LDAT_ACT=LCPDAT304
FDAT_ACT=Ffred5codoD
BAS(#CP_PARAMS,0.1)
LIN Xfred5codoD
;ENDFOLD

;--- Abrir gripper ---
$OUT[101] = TRUE
$OUT[102] = FALSE
WAIT SEC 1

;FOLD LIN fred6codoDA Vel=2 m/s CPDAT306 Tool[1]:navaja Base[0];%{PE}%R 8.3.40,%MKUKATPBASIS,%CMOVE,%VLIN,%P 1:LIN, 2:fred6codoDA, 3:, 5:2, 7:CPDAT306
$BWDSTART=FALSE
LDAT_ACT=LCPDAT306
FDAT_ACT=Ffred6codoDA
BAS(#CP_PARAMS,2)
LIN Xfred6codoDA
;ENDFOLD

;--- Movimiento a centro ---
PDAT_ACT=PPDAT4
FDAT_ACT=Fcentro
BAS(#PTP_PARAMS,20)
PTP Xcentro

;PERFILIZQUIERDO4 ARRIBA
$BWDSTART=FALSE
LDAT_ACT=LCPDAT204
FDAT_ACT=Ffred4PIA
BAS(#CP_PARAMS,2)
LIN Xfred4PIA


;PERFILIZQUIERDO4 ABAJO
$BWDSTART=FALSE
LDAT_ACT=LCPDAT203
FDAT_ACT=Ffred4PI
BAS(#CP_PARAMS,2)
LIN Xfred4PI

;--- Cerrar gripper ---
$OUT[101] = FALSE
$OUT[102] = TRUE
WAIT SEC 1

;PERFILIZQUIERDO4 ARRIBA
$BWDSTART=FALSE
LDAT_ACT=LCPDAT206
FDAT_ACT=Ffred4PIA_1
BAS(#CP_PARAMS,2)
LIN Xfred4PIA_1



;FOLD LIN fred4PIIA Vel=2 m/s CPDAT267 Tool[1]:navaja Base[0];%{PE}%R 8.3.40,%MKUKATPBASIS,%CMOVE,%VLIN,%P 1:LIN, 2:fred4PIIA, 3:, 5:2, 7:CPDAT267
$BWDSTART=FALSE
LDAT_ACT=LCPDAT267
FDAT_ACT=Ffred4PIIA
BAS(#CP_PARAMS,2)
LIN Xfred4PIIA
;ENDFOLD



;FOLD LIN fred4PII Vel=2 m/s CPDAT266 Tool[1]:navaja Base[0];%{PE}%R 8.3.40,%MKUKATPBASIS,%CMOVE,%VLIN,%P 1:LIN, 2:fred4PII, 3:, 5:2, 7:CPDAT266
$BWDSTART=FALSE
LDAT_ACT=LCPDAT266
FDAT_ACT=Ffred4PII
BAS(#CP_PARAMS,0.1)
LIN Xfred4PII
;ENDFOLD

;--- Abrir gripper ---
$OUT[101] = TRUE
$OUT[102] = FALSE
WAIT SEC 1

;FOLD LIN fred4PIIA_2 Vel=2 m/s CPDAT267 Tool[1]:navaja Base[0];%{PE}%R 8.3.40,%MKUKATPBASIS,%CMOVE,%VLIN,%P 1:LIN, 2:fred4PIIA_2, 3:, 5:2, 7:CPDAT267
$BWDSTART=FALSE
LDAT_ACT=LCPDAT276
FDAT_ACT=Ffred4PIIA_2
BAS(#CP_PARAMS,0.1)
LIN Xfred4PIIA_2
;ENDFOLD


;PERFILDERECHO4 ARRIBA
$BWDSTART=FALSE
PDAT_ACT=PPDAT46
FDAT_ACT=Ffred4PDA
BAS(#PTP_PARAMS,20)
PTP Xfred4PDA

;PERFILDERECHO4 ABAJO
$BWDSTART=FALSE
LDAT_ACT=LCPDAT205
FDAT_ACT=Ffred4PD
BAS(#CP_PARAMS,2)
LIN Xfred4PD


;--- Cerrar gripper ---
$OUT[101] = FALSE
$OUT[102] = TRUE
WAIT SEC 1

;PERFILDERECHO4 ARRIBA
$BWDSTART=FALSE
PDAT_ACT=PPDAT47
FDAT_ACT=Ffred4PDA_1
BAS(#PTP_PARAMS,20)
PTP Xfred4PDA_1



;FOLD LIN fred44PDA Vel=2 m/s CPDAT269 Tool[1]:navaja Base[0];%{PE}%R 8.3.40,%MKUKATPBASIS,%CMOVE,%VLIN,%P 1:LIN, 2:fred44PDA, 3:, 5:2, 7:CPDAT269
$BWDSTART=FALSE
LDAT_ACT=LCPDAT269
FDAT_ACT=Ffred44PDA
BAS(#CP_PARAMS,2)
LIN Xfred44PDA
;ENDFOLD


;FOLD LIN fred4PDD Vel=2 m/s CPDAT268 Tool[1]:navaja Base[0];%{PE}%R 8.3.40,%MKUKATPBASIS,%CMOVE,%VLIN,%P 1:LIN, 2:fred4PDD, 3:, 5:2, 7:CPDAT268
$BWDSTART=FALSE
LDAT_ACT=LCPDAT268
FDAT_ACT=Ffred4PDD
BAS(#CP_PARAMS,0.1)
LIN Xfred4PDD
;ENDFOLD

;--- Abrir gripper ---
$OUT[101] = TRUE
$OUT[102] = FALSE
WAIT SEC 1


;FOLD LIN fred44PDA_1 Vel=2 m/s CPDAT269 Tool[1]:navaja Base[0];%{PE}%R 8.3.40,%MKUKATPBASIS,%CMOVE,%VLIN,%P 1:LIN, 2:fred44PDA_1, 3:, 5:2, 7:CPDAT269
$BWDSTART=FALSE
LDAT_ACT=LCPDAT277
FDAT_ACT=Ffred44PDA_1
BAS(#CP_PARAMS,0.1)
LIN Xfred44PDA_1
;ENDFOLD


;--- Movimiento a centro ---
PDAT_ACT=PPDAT4
FDAT_ACT=Fcentro
BAS(#PTP_PARAMS,20)
PTP Xcentro


;FOLD LIN fred44ventA Vel=2 m/s CPDAT282 Tool[1]:navaja Base[0];%{PE}%R 8.3.40,%MKUKATPBASIS,%CMOVE,%VLIN,%P 1:LIN, 2:fred44ventA, 3:, 5:2, 7:CPDAT282
$BWDSTART=FALSE
LDAT_ACT=LCPDAT282
FDAT_ACT=Ffred44ventA
BAS(#CP_PARAMS,2)
LIN Xfred44ventA
;ENDFOLD

;FOLD LIN fred44vent Vel=2 m/s CPDAT281 Tool[1]:navaja Base[0];%{PE}%R 8.3.40,%MKUKATPBASIS,%CMOVE,%VLIN,%P 1:LIN, 2:fred44vent, 3:, 5:2, 7:CPDAT281
$BWDSTART=FALSE
LDAT_ACT=LCPDAT281
FDAT_ACT=Ffred44vent
BAS(#CP_PARAMS,2)
LIN Xfred44vent
;ENDFOLD

;--- Cerrar gripper ---
$OUT[101] = FALSE
$OUT[102] = TRUE
WAIT SEC 1

;FOLD LIN fred44ventA_2 Vel=2 m/s CPDAT282 Tool[1]:navaja Base[0];%{PE}%R 8.3.40,%MKUKATPBASIS,%CMOVE,%VLIN,%P 1:LIN, 2:fred44ventA_2, 3:, 5:2, 7:CPDAT282
$BWDSTART=FALSE
LDAT_ACT=LCPDAT295
FDAT_ACT=Ffred44ventA_2
BAS(#CP_PARAMS,2)
LIN Xfred44ventA_2
;ENDFOLD

;--- Movimiento a vent88 ---
PDAT_ACT=PPDAT18
FDAT_ACT=Fvent88
BAS(#PTP_PARAMS,2)
PTP Xvent88


;FOLD LIN vent4fredA Vel=2 m/s CPDAT303 Tool[1]:navaja Base[0];%{PE}%R 8.3.40,%MKUKATPBASIS,%CMOVE,%VLIN,%P 1:LIN, 2:vent4fredA, 3:, 5:2, 7:CPDAT303
$BWDSTART=FALSE
LDAT_ACT=LCPDAT303
FDAT_ACT=Fvent4fredA
BAS(#CP_PARAMS,2)
LIN Xvent4fredA
;ENDFOLD

;FOLD LIN ven4fredP Vel=2 m/s CPDAT283 Tool[1]:navaja Base[0];%{PE}%R 8.3.40,%MKUKATPBASIS,%CMOVE,%VLIN,%P 1:LIN, 2:ven4fredP, 3:, 5:2, 7:CPDAT283
$BWDSTART=FALSE
LDAT_ACT=LCPDAT283
FDAT_ACT=Fven4fredP
BAS(#CP_PARAMS,0.02)
LIN Xven4fredP
;ENDFOLD

;--- Abrir gripper ---
$OUT[101] = TRUE
$OUT[102] = FALSE
WAIT SEC 1


;FOLD LIN vent4fredA_1 Vel=2 m/s CPDAT302 Tool[1]:navaja Base[0];%{PE}%R 8.3.40,%MKUKATPBASIS,%CMOVE,%VLIN,%P 1:LIN, 2:vent4fredA_1, 3:, 5:2, 7:CPDAT302
$BWDSTART=FALSE
LDAT_ACT=LCPDAT302
FDAT_ACT=Fvent4fredA_1
BAS(#CP_PARAMS,2)
LIN Xvent4fredA_1
;ENDFOLD

;--- Movimiento final a centro ---
PDAT_ACT=PPDAT4
FDAT_ACT=Fcentro
BAS(#PTP_PARAMS,20)
PTP Xcentro


;---------------------------------------------------------------------------------------------------------------------------------------------------------
;FRED 5;---------------------------------------------------------------------------------------------------------------------------------------------------------

$OUT[101] = FALSE
WAIT SEC 0.5

;--- Movimiento a centro con velocidad reducida ---
PDAT_ACT=PPDAT4
FDAT_ACT=Fcentro
BAS(#PTP_PARAMS,20)
PTP Xcentro

;--- Abrir gripper ---
$OUT[101] = TRUE
$OUT[102] = FALSE
WAIT SEC 1

;--- Movimiento a codoIB3 ---
LDAT_ACT=LCPDAT2
FDAT_ACT=FcodoIB3
BAS(#CP_PARAMS,10)
LIN XcodoIB3

;--- Movimiento a codoIB2 ---
LDAT_ACT=LCPDAT5
FDAT_ACT=FcodoIB2
BAS(#CP_PARAMS,10)
LIN XcodoIB2


$BWDSTART=FALSE
LDAT_ACT=LCPDAT45
FDAT_ACT=FIB3
BAS(#CP_PARAMS,2)
LIN XIB3



;--- Cerrar gripper ---
$OUT[101] = FALSE
$OUT[102] = TRUE
WAIT SEC 1

;--- Regreso por codoIB2 ---
LDAT_ACT=LCPDAT5
FDAT_ACT=FcodoIB2
BAS(#CP_PARAMS,10)
LIN XcodoIB2

;--- Regreso por codoIB3 ---
LDAT_ACT=LCPDAT2
FDAT_ACT=FcodoIB3
BAS(#CP_PARAMS,10)
LIN XcodoIB3

;--- Regreso a centro ---
PDAT_ACT=PPDAT4
FDAT_ACT=Fcentro
BAS(#PTP_PARAMS,20)
PTP Xcentro


$BWDSTART=FALSE
LDAT_ACT=LCPDAT47
FDAT_ACT=FIP3
BAS(#CP_PARAMS,2)
LIN XIP3


$BWDSTART=FALSE
LDAT_ACT=LCPDAT46
FDAT_ACT=FIP2
BAS(#CP_PARAMS,0.1)
LIN XIP2


;--- Abrir gripper ---
$OUT[101] = TRUE
$OUT[102] = FALSE
WAIT SEC 1


$BWDSTART=FALSE
LDAT_ACT=LCPDAT60
FDAT_ACT=FIP4
BAS(#CP_PARAMS,0.1)
LIN XIP4



;--- Movimiento a centro ---
PDAT_ACT=PPDAT4
FDAT_ACT=Fcentro
BAS(#PTP_PARAMS,20)
PTP Xcentro

;--- Movimiento a codoD2 ---
PDAT_ACT=PPDAT6
FDAT_ACT=FcodoD2
BAS(#PTP_PARAMS,20)
PTP XcodoD2


$BWDSTART=FALSE
LDAT_ACT=LCPDAT66
FDAT_ACT=FcodoD4
BAS(#CP_PARAMS,2)
LIN XcodoD4


;--- Cerrar gripper ---
$OUT[101] = FALSE
$OUT[102] = TRUE
WAIT SEC 1


$BWDSTART=FALSE
LDAT_ACT=LCPDAT68
FDAT_ACT=FcodoDD5
BAS(#CP_PARAMS,2)
LIN XcodoDD5


;--- Movimiento a centro_5 con velocidad reducida ---
PDAT_ACT=PPDAT20
FDAT_ACT=Fcentro_5
BAS(#PTP_PARAMS,20)
PTP Xcentro_5




;FOLD LIN fred55codoDA Vel=2 m/s CPDAT308 Tool[1]:navaja Base[0];%{PE}%R 8.3.40,%MKUKATPBASIS,%CMOVE,%VLIN,%P 1:LIN, 2:fred55codoDA, 3:, 5:2, 7:CPDAT308
$BWDSTART=FALSE
LDAT_ACT=LCPDAT308
FDAT_ACT=Ffred55codoDA
BAS(#CP_PARAMS,2)
LIN Xfred55codoDA
;ENDFOLD

;FOLD LIN fred55codoD Vel=2 m/s CPDAT307 Tool[1]:navaja Base[0];%{PE}%R 8.3.40,%MKUKATPBASIS,%CMOVE,%VLIN,%P 1:LIN, 2:fred55codoD, 3:, 5:2, 7:CPDAT307
$BWDSTART=FALSE
LDAT_ACT=LCPDAT307
FDAT_ACT=Ffred55codoD
BAS(#CP_PARAMS,0.1)
LIN Xfred55codoD
;ENDFOLD

;--- Abrir gripper ---
$OUT[101] = TRUE
$OUT[102] = FALSE
WAIT SEC 1


;FOLD LIN fred55codoDAA Vel=2 m/s CPDAT309 Tool[1]:navaja Base[0];%{PE}%R 8.3.40,%MKUKATPBASIS,%CMOVE,%VLIN,%P 1:LIN, 2:fred55codoDAA, 3:, 5:2, 7:CPDAT309
$BWDSTART=FALSE
LDAT_ACT=LCPDAT309
FDAT_ACT=Ffred55codoDAA
BAS(#CP_PARAMS,2)
LIN Xfred55codoDAA
;ENDFOLD
;--- Movimiento a centro ---
PDAT_ACT=PPDAT4
FDAT_ACT=Fcentro
BAS(#PTP_PARAMS,20)
PTP Xcentro

;PERFIFLIZQUIERDO5 ARRIBA
;FOLD PTP fred56PIA Vel=100 % PDAT59 Tool[1]:navaja Base[0];%{PE}%R 8.3.40,%MKUKATPBASIS,%CMOVE,%VPTP,%P 1:PTP, 2:fred56PIA, 3:, 5:100, 7:PDAT59
$BWDSTART=FALSE
PDAT_ACT=PPDAT59
FDAT_ACT=Ffred56PIA
BAS(#PTP_PARAMS,20)
PTP Xfred56PIA
;ENDFOLD

;PERFILIZQUIERDO5 ABAJO
;FOLD LIN fred55PI Vel=2 m/s CPDAT270 Tool[1]:navaja Base[0];%{PE}%R 8.3.40,%MKUKATPBASIS,%CMOVE,%VLIN,%P 1:LIN, 2:fred55PI, 3:, 5:2, 7:CPDAT270
$BWDSTART=FALSE
LDAT_ACT=LCPDAT270
FDAT_ACT=Ffred55PI
BAS(#CP_PARAMS,2)
LIN Xfred55PI
;ENDFOLD

;--- Cerrar gripper ---
$OUT[101] = FALSE
$OUT[102] = TRUE
WAIT SEC 1

;PERFIFLIZQUIERDO5 ARRIBA
;FOLD PTP fred56PIA_2 Vel=100 % PDAT61 Tool[1]:navaja Base[0];%{PE}%R 8.3.40,%MKUKATPBASIS,%CMOVE,%VPTP,%P 1:PTP, 2:fred56PIA_2, 3:, 5:100, 7:PDAT61
$BWDSTART=FALSE
PDAT_ACT=PPDAT61
FDAT_ACT=Ffred56PIA_2
BAS(#PTP_PARAMS,20)
PTP Xfred56PIA_2
;ENDFOLD

;FOLD LIN fred55PIIAA Vel=2 m/s CPDAT298 Tool[1]:navaja Base[0];%{PE}%R 8.3.40,%MKUKATPBASIS,%CMOVE,%VLIN,%P 1:LIN, 2:fred55PIIAA, 3:, 5:2, 7:CPDAT298
$BWDSTART=FALSE
LDAT_ACT=LCPDAT298
FDAT_ACT=Ffred55PIIAA
BAS(#CP_PARAMS,2)
LIN Xfred55PIIAA
;ENDFOLD

;FOLD LIN fred55PIp Vel=2 m/s CPDAT297 Tool[1]:navaja Base[0];%{PE}%R 8.3.40,%MKUKATPBASIS,%CMOVE,%VLIN,%P 1:LIN, 2:fred55PIp, 3:, 5:2, 7:CPDAT297
$BWDSTART=FALSE
LDAT_ACT=LCPDAT297
FDAT_ACT=Ffred55PIp
BAS(#CP_PARAMS,0.1)
LIN Xfred55PIp
;ENDFOLD

;--- Abrir gripper ---
$OUT[101] = TRUE
$OUT[102] = FALSE
WAIT SEC 1

;FOLD LIN fred55PIIAA Vel=2 m/s CPDAT298 Tool[1]:navaja Base[0];%{PE}%R 8.3.40,%MKUKATPBASIS,%CMOVE,%VLIN,%P 1:LIN, 2:fred55PIIAA, 3:, 5:2, 7:CPDAT298
$BWDSTART=FALSE
LDAT_ACT=LCPDAT298
FDAT_ACT=Ffred55PIIAA
BAS(#CP_PARAMS,0.1)
LIN Xfred55PIIAA
;ENDFOLD


;FOLD LIN fred55PIIAA Vel=2 m/s CPDAT298 Tool[1]:navaja Base[0];%{PE}%R 8.3.40,%MKUKATPBASIS,%CMOVE,%VLIN,%P 1:LIN, 2:fred55PIIAA, 3:, 5:2, 7:CPDAT298
$BWDSTART=FALSE
LDAT_ACT=LCPDAT298
FDAT_ACT=Ffred55PIIAA
BAS(#CP_PARAMS,2)
LIN Xfred55PIIAA
;ENDFOLD

;PERFILDERECHO5 ABAJO

;FOLD LIN fred5PDDA Vel=2 m/s CPDAT301 Tool[1]:navaja Base[0];%{PE}%R 8.3.40,%MKUKATPBASIS,%CMOVE,%VLIN,%P 1:LIN, 2:fred5PDDA, 3:, 5:2, 7:CPDAT301
$BWDSTART=FALSE
LDAT_ACT=LCPDAT301
FDAT_ACT=Ffred5PDDA
BAS(#CP_PARAMS,2)
LIN Xfred5PDDA
;ENDFOLD

;FOLD LIN fred5PDDD Vel=2 m/s CPDAT300 Tool[1]:navaja Base[0];%{PE}%R 8.3.40,%MKUKATPBASIS,%CMOVE,%VLIN,%P 1:LIN, 2:fred5PDDD, 3:, 5:2, 7:CPDAT300
$BWDSTART=FALSE
LDAT_ACT=LCPDAT300
FDAT_ACT=Ffred5PDDD
BAS(#CP_PARAMS,2)
LIN Xfred5PDDD
;ENDFOLD


;--- Cerrar gripper ---
$OUT[101] = FALSE
$OUT[102] = TRUE
WAIT SEC 1

;FOLD LIN fred5PDDA Vel=2 m/s CPDAT301 Tool[1]:navaja Base[0];%{PE}%R 8.3.40,%MKUKATPBASIS,%CMOVE,%VLIN,%P 1:LIN, 2:fred5PDDA, 3:, 5:2, 7:CPDAT301
$BWDSTART=FALSE
LDAT_ACT=LCPDAT301
FDAT_ACT=Ffred5PDDA
BAS(#CP_PARAMS,2)
LIN Xfred5PDDA
;ENDFOLD



;FOLD LIN fred5PDAA Vel=2 m/s CPDAT272 Tool[1]:navaja Base[0];%{PE}%R 8.3.40,%MKUKATPBASIS,%CMOVE,%VLIN,%P 1:LIN, 2:fred5PDAA, 3:, 5:2, 7:CPDAT272
$BWDSTART=FALSE
LDAT_ACT=LCPDAT272
FDAT_ACT=Ffred5PDAA
BAS(#CP_PARAMS,2)
LIN Xfred5PDAA
;ENDFOLD


;FOLD LIN fred5PIP Vel=2 m/s CPDAT271 Tool[1]:navaja Base[0];%{PE}%R 8.3.40,%MKUKATPBASIS,%CMOVE,%VLIN,%P 1:LIN, 2:fred5PIP, 3:, 5:2, 7:CPDAT271
$BWDSTART=FALSE
LDAT_ACT=LCPDAT271
FDAT_ACT=Ffred5PIP
BAS(#CP_PARAMS,0.1)
LIN Xfred5PIP
;ENDFOLD
;--- Abrir gripper ---
$OUT[101] = TRUE
$OUT[102] = FALSE
WAIT SEC 1

;FOLD LIN fred5PDAA_1 Vel=2 m/s CPDAT272 Tool[1]:navaja Base[0];%{PE}%R 8.3.40,%MKUKATPBASIS,%CMOVE,%VLIN,%P 1:LIN, 2:fred5PDAA_1, 3:, 5:2, 7:CPDAT272
$BWDSTART=FALSE
LDAT_ACT=LCPDAT278
FDAT_ACT=Ffred5PDAA_1
BAS(#CP_PARAMS,0.1)
LIN Xfred5PDAA_1
;ENDFOLD


;--- Movimiento a centro ---
PDAT_ACT=PPDAT4
FDAT_ACT=Fcentro
BAS(#PTP_PARAMS,20)
PTP Xcentro

;FOLD LIN ventfred5A Vel=2 m/s CPDAT287 Tool[1]:navaja Base[0];%{PE}%R 8.3.40,%MKUKATPBASIS,%CMOVE,%VLIN,%P 1:LIN, 2:ventfred5A, 3:, 5:2, 7:CPDAT287
$BWDSTART=FALSE
LDAT_ACT=LCPDAT287
FDAT_ACT=Fventfred5A
BAS(#CP_PARAMS,2)
LIN Xventfred5A
;ENDFOLD

;FOLD LIN ventfred5 Vel=2 m/s CPDAT286 Tool[1]:navaja Base[0];%{PE}%R 8.3.40,%MKUKATPBASIS,%CMOVE,%VLIN,%P 1:LIN, 2:ventfred5, 3:, 5:2, 7:CPDAT286
$BWDSTART=FALSE
LDAT_ACT=LCPDAT286
FDAT_ACT=Fventfred5
BAS(#CP_PARAMS,2)
LIN Xventfred5
;ENDFOLD

;--- Cerrar gripper ---
$OUT[101] = FALSE
$OUT[102] = TRUE
WAIT SEC 1

;FOLD LIN ventfred5A_1 Vel=2 m/s CPDAT287 Tool[1]:navaja Base[0];%{PE}%R 8.3.40,%MKUKATPBASIS,%CMOVE,%VLIN,%P 1:LIN, 2:ventfred5A_1, 3:, 5:2, 7:CPDAT287
$BWDSTART=FALSE
LDAT_ACT=LCPDAT296
FDAT_ACT=Fventfred5A_1
BAS(#CP_PARAMS,2)
LIN Xventfred5A_1
;ENDFOLD

;--- Movimiento a vent88 ---
PDAT_ACT=PPDAT18
FDAT_ACT=Fvent88
BAS(#PTP_PARAMS,2)
PTP Xvent88


;FOLD LIN fred5VENTTa Vel=2 m/s CPDAT274 Tool[1]:navaja Base[0];%{PE}%R 8.3.40,%MKUKATPBASIS,%CMOVE,%VLIN,%P 1:LIN, 2:fred5VENTTa, 3:, 5:2, 7:CPDAT274
$BWDSTART=FALSE
LDAT_ACT=LCPDAT274
FDAT_ACT=Ffred5VENTTa
BAS(#CP_PARAMS,2)
LIN Xfred5VENTTa
;ENDFOLD

;FOLD LIN fred5VENTT Vel=2 m/s CPDAT273 Tool[1]:navaja Base[0];%{PE}%R 8.3.40,%MKUKATPBASIS,%CMOVE,%VLIN,%P 1:LIN, 2:fred5VENTT, 3:, 5:2, 7:CPDAT273
$BWDSTART=FALSE
LDAT_ACT=LCPDAT273
FDAT_ACT=Ffred5VENTT
BAS(#CP_PARAMS,0.02)
LIN Xfred5VENTT
;ENDFOLD

;--- Abrir gripper ---
$OUT[101] = TRUE
$OUT[102] = FALSE
WAIT SEC 1

;FOLD LIN fred5VENTTa_2 Vel=2 m/s CPDAT274 Tool[1]:navaja Base[0];%{PE}%R 8.3.40,%MKUKATPBASIS,%CMOVE,%VLIN,%P 1:LIN, 2:fred5VENTTa_2, 3:, 5:2, 7:CPDAT274
$BWDSTART=FALSE
LDAT_ACT=LCPDAT280
FDAT_ACT=Ffred5VENTTa_2
BAS(#CP_PARAMS,2)
LIN Xfred5VENTTa_2
;ENDFOLD

;--- Movimiento final a centro ---
PDAT_ACT=PPDAT4
FDAT_ACT=Fcentro
BAS(#PTP_PARAMS,20)
PTP Xcentro



ENDFOR

INTERRUPT OFF 25
$OUT[105]=TRUE

END

DEF PAUSA()

BRAKE

WAIT FOR ($IN[107])

END

--- FrED_Main.dat ---
&ACCESS RVO
DEFDAT codigoWS3
;FOLD EXTERNAL DECLARATIONS;%{PE}%MKUKATPBASIS,%CEXT,%VCOMMON,%P
;FOLD GRIPPERTECH EXT
EXT  H50 (INT  :IN,INT  :IN,INT  :IN,GRP_TYP  :IN )
;ENDFOLD (GRIPPERTECH EXT)
;FOLD SPOTTECH EXT
EXT  USERSPOT (S_COMMAND  :IN,SPOT_TYPE  :IN )
;ENDFOLD (SPOTTECH EXT)
;FOLD BASISTECH EXT;%{PE}%MKUKATPBASIS,%CEXT,%VEXT,%P
EXT  BAS (BAS_COMMAND  :IN,REAL  :IN )
DECL INT SUCCESS
;ENDFOLD (BASISTECH EXT)
;FOLD USER EXT;%{E}%MKUKATPUSER,%CEXT,%VEXT,%P
;Make your modifications here

;ENDFOLD (USER EXT)
;ENDFOLD (EXTERNAL DECLARATIONS)
DECL BASIS_SUGG_T LAST_BASIS={POINT1[] "fred55codoDAA           ",POINT2[] "fred55codoDAA           ",CP_PARAMS[] "CPDAT309                ",PTP_PARAMS[] "PDAT63                  ",CONT[] "                        ",CP_VEL[] "2                       ",PTP_VEL[] "100                     ",SYNC_PARAMS[] "SYNCDAT                 ",SPL_NAME[] "S0                      ",A_PARAMS[] "ADAT0                   "}
DECL E6POS XP1={X 341.825592,Y 43.2718811,Z 440.001526,A -60.3082466,B 16.7546577,C -168.888596,S 2,T 10,E1 0.0,E2 0.0,E3 0.0,E4 0.0,E5 0.0,E6 0.0}
DECL FDAT FP1={TOOL_NO 1,BASE_NO 0,IPO_FRAME #BASE,POINT2[] " ",TQ_STATE FALSE}
DECL PDAT PPDAT1={VEL 100.000,ACC 100.000,APO_DIST 100.000,APO_MODE #CDIS,GEAR_JERK 50.0000,EXAX_IGN 0}
DECL E6POS XCODOIB={X 169.580139,Y 270.518555,Z 98.2024536,A -5.40927553,B 17.7038708,C -156.222351,S 2,T 11,E1 0.0,E2 0.0,E3 0.0,E4 0.0,E5 0.0,E6 0.0}
DECL FDAT FcodoIB={TOOL_NO 1,BASE_NO 0,IPO_FRAME #BASE,POINT2[] " ",TQ_STATE FALSE}
DECL LDAT LCPDAT1={VEL 2.00000,ACC 100.000,APO_DIST 100.000,APO_FAC 50.0000,AXIS_VEL 100.000,AXIS_ACC 100.000,ORI_TYP #VAR,CIRC_TYP #BASE,JERK_FAC 50.0000,GEAR_JERK 50.0000,EXAX_IGN 0}
DECL PDAT PPDAT2={VEL 100.000,ACC 100.000,APO_DIST 100.000,APO_MODE #CDIS,GEAR_JERK 50.0000,EXAX_IGN 0}
DECL E6POS XCODOIB2={X 169.370163,Y 288.233887,Z 215.088318,A -9.98564243,B -1.58595812,C 179.083130,S 2,T 3,E1 0.0,E2 0.0,E3 0.0,E4 0.0,E5 0.0,E6 0.0}
DECL FDAT FcodoIB2={TOOL_NO 1,BASE_NO 0,IPO_FRAME #BASE,POINT2[] " ",TQ_STATE FALSE}
DECL PDAT PPDAT3={VEL 100.000,ACC 100.000,APO_DIST 100.000,APO_MODE #CDIS,GEAR_JERK 50.0000,EXAX_IGN 0}
DECL E6POS XCODOIB3={X 169.372009,Y 288.237305,Z 503.685242,A -9.98564529,B -1.58597386,C 179.083130,S 2,T 3,E1 0.0,E2 0.0,E3 0.0,E4 0.0,E5 0.0,E6 0.0}
DECL FDAT FcodoIB3={TOOL_NO 1,BASE_NO 0,IPO_FRAME #BASE,POINT2[] " ",TQ_STATE FALSE}
DECL LDAT LCPDAT2={VEL 2.00000,ACC 100.000,APO_DIST 100.000,APO_FAC 50.0000,AXIS_VEL 100.000,AXIS_ACC 100.000,ORI_TYP #VAR,CIRC_TYP #BASE,JERK_FAC 50.0000,GEAR_JERK 50.0000,EXAX_IGN 0}
DECL E6POS XCENTRO={X 222.017685,Y 1.93147576,Z 503.686340,A 38.9071503,B -1.58586597,C 179.083191,S 2,T 10,E1 0.0,E2 0.0,E3 0.0,E4 0.0,E5 0.0,E6 0.0}
DECL FDAT Fcentro={TOOL_NO 1,BASE_NO 0,IPO_FRAME #BASE,POINT2[] " ",TQ_STATE FALSE}
DECL PDAT PPDAT4={VEL 100.000,ACC 100.000,APO_DIST 100.000,APO_MODE #CDIS,GEAR_JERK 50.0000,EXAX_IGN 0}
DECL E6POS XCODOIP={X 495.259338,Y -72.1194916,Z 105.335014,A 42.5121155,B -1.58614099,C 179.082733,S 2,T 10,E1 0.0,E2 0.0,E3 0.0,E4 0.0,E5 0.0,E6 0.0}
DECL FDAT FcodoIP={TOOL_NO 1,BASE_NO 0,IPO_FRAME #BASE,POINT2[] " ",TQ_STATE FALSE}
DECL LDAT LCPDAT3={VEL 2.00000,ACC 100.000,APO_DIST 100.000,APO_FAC 50.0000,AXIS_VEL 100.000,AXIS_ACC 100.000,ORI_TYP #VAR,CIRC_TYP #BASE,JERK_FAC 50.0000,GEAR_JERK 50.0000,EXAX_IGN 0}
DECL E6POS XCODOIPA={X 495.277374,Y -72.1219254,Z 305.970398,A 42.5108,B -1.58776,C 179.080200,S 2,T 10,E1 0.0,E2 0.0,E3 0.0,E4 0.0,E5 0.0,E6 0.0}
DECL FDAT FcodoIPA={TOOL_NO 1,BASE_NO 0,IPO_FRAME #BASE,POINT2[] " ",TQ_STATE FALSE}
DECL PDAT PPDAT5={VEL 100.000,ACC 100.000,APO_DIST 100.000,APO_MODE #CDIS,GEAR_JERK 50.0000,EXAX_IGN 0}
DECL LDAT LCPDAT4={VEL 2.00000,ACC 100.000,APO_DIST 100.000,APO_FAC 50.0000,AXIS_VEL 100.000,AXIS_ACC 100.000,ORI_TYP #VAR,CIRC_TYP #BASE,JERK_FAC 50.0000,GEAR_JERK 50.0000,EXAX_IGN 0}
DECL LDAT LCPDAT5={VEL 2.00000,ACC 100.000,APO_DIST 100.000,APO_FAC 50.0000,AXIS_VEL 100.000,AXIS_ACC 100.000,ORI_TYP #VAR,CIRC_TYP #BASE,JERK_FAC 50.0000,GEAR_JERK 50.0000,EXAX_IGN 0}
DECL E6POS XCODOD={X 120.584869,Y 330.035919,Z 251.804016,A -5.40004730,B 17.7066059,C -156.192,S 2,T 11,E1 0.0,E2 0.0,E3 0.0,E4 0.0,E5 0.0,E6 0.0}
DECL FDAT FcodoD={TOOL_NO 1,BASE_NO 0,IPO_FRAME #BASE,POINT2[] " ",TQ_STATE FALSE}
DECL LDAT LCPDAT6={VEL 2.00000,ACC 100.000,APO_DIST 100.000,APO_FAC 50.0000,AXIS_VEL 100.000,AXIS_ACC 100.000,ORI_TYP #VAR,CIRC_TYP #BASE,JERK_FAC 50.0000,GEAR_JERK 50.0000,EXAX_IGN 0}
DECL E6POS XCODOD2={X 120.584869,Y 330.035919,Z 422.057,A -5.40004730,B 17.7066059,C -156.192,S 2,T 11,E1 0.0,E2 0.0,E3 0.0,E4 0.0,E5 0.0,E6 0.0}
DECL FDAT FcodoD2={TOOL_NO 1,BASE_NO 0,IPO_FRAME #BASE,POINT2[] " ",TQ_STATE FALSE}
DECL PDAT PPDAT6={VEL 100.000,ACC 100.000,APO_DIST 100.000,APO_MODE #CDIS,GEAR_JERK 50.0000,EXAX_IGN 0}
DECL E6POS XCODODP={X 495.551361,Y 75.4896164,Z 104.322121,A 42.5106506,B -1.61344421,C 179.062820,S 2,T 11,E1 0.0,E2 0.0,E3 0.0,E4 0.0,E5 0.0,E6 0.0}
DECL FDAT FcodoDP={TOOL_NO 1,BASE_NO 0,IPO_FRAME #BASE,POINT2[] " ",TQ_STATE FALSE}
DECL LDAT LCPDAT7={VEL 2.00000,ACC 100.000,APO_DIST 100.000,APO_FAC 50.0000,AXIS_VEL 100.000,AXIS_ACC 100.000,ORI_TYP #VAR,CIRC_TYP #BASE,JERK_FAC 50.0000,GEAR_JERK 50.0000,EXAX_IGN 0}
DECL E6POS XCODODPA={X 495.551361,Y 75.4896164,Z 295.991516,A 42.5106506,B -1.61344421,C 179.062820,S 2,T 11,E1 0.0,E2 0.0,E3 0.0,E4 0.0,E5 0.0,E6 0.0}
DECL FDAT FcodoDPA={TOOL_NO 1,BASE_NO 0,IPO_FRAME #BASE,POINT2[] " ",TQ_STATE FALSE}
DECL PDAT PPDAT7={VEL 100.000,ACC 100.000,APO_DIST 100.000,APO_MODE #CDIS,GEAR_JERK 50.0000,EXAX_IGN 0}
DECL E6POS XPI={X 488.794952,Y 263.522217,Z 330.558746,A 38.9071503,B -1.58586621,C 179.083191,S 2,T 3,E1 0.0,E2 0.0,E3 0.0,E4 0.0,E5 0.0,E6 0.0}
DECL FDAT FPI={TOOL_NO 1,BASE_NO 0,IPO_FRAME #BASE,POINT2[] " ",TQ_STATE FALSE}
DECL LDAT LCPDAT8={VEL 2.00000,ACC 100.000,APO_DIST 100.000,APO_FAC 50.0000,AXIS_VEL 100.000,AXIS_ACC 100.000,ORI_TYP #VAR,CIRC_TYP #BASE,JERK_FAC 50.0000,GEAR_JERK 50.0000,EXAX_IGN 0}
DECL E6POS XPIA={X 488.794952,Y 263.522217,Z 467.844391,A 38.9071503,B -1.58586633,C 179.083191,S 2,T 3,E1 0.0,E2 0.0,E3 0.0,E4 0.0,E5 0.0,E6 0.0}
DECL FDAT FPIA={TOOL_NO 1,BASE_NO 0,IPO_FRAME #BASE,POINT2[] " ",TQ_STATE FALSE}
DECL LDAT LCPDAT9={VEL 2.00000,ACC 100.000,APO_DIST 100.000,APO_FAC 50.0000,AXIS_VEL 100.000,AXIS_ACC 100.000,ORI_TYP #VAR,CIRC_TYP #BASE,JERK_FAC 50.0000,GEAR_JERK 50.0000,EXAX_IGN 0}
DECL E6POS XPIP={X 503.498657,Y -68.2245560,Z 339.513977,A 43.3322525,B -1.62203932,C 179.037308,S 2,T 10,E1 0.0,E2 0.0,E3 0.0,E4 0.0,E5 0.0,E6 0.0}
DECL FDAT Fpip={TOOL_NO 1,BASE_NO 0,IPO_FRAME #BASE,POINT2[] " ",TQ_STATE FALSE}
DECL LDAT LCPDAT10={VEL 2.00000,ACC 100.000,APO_DIST 100.000,APO_FAC 50.0000,AXIS_VEL 100.000,AXIS_ACC 100.000,ORI_TYP #VAR,CIRC_TYP #BASE,JERK_FAC 50.0000,GEAR_JERK 50.0000,EXAX_IGN 0}
DECL E6POS XPIPA={X 503.395630,Y -68.2099609,Z 442.073,A 43.3303375,B -1.60676658,C 179.056412,S 2,T 10,E1 0.0,E2 0.0,E3 0.0,E4 0.0,E5 0.0,E6 0.0}
DECL FDAT Fpipa={TOOL_NO 1,BASE_NO 0,IPO_FRAME #BASE,POINT2[] " ",TQ_STATE FALSE}
DECL LDAT LCPDAT11={VEL 2.00000,ACC 100.000,APO_DIST 100.000,APO_FAC 50.0000,AXIS_VEL 100.000,AXIS_ACC 100.000,ORI_TYP #VAR,CIRC_TYP #BASE,JERK_FAC 50.0000,GEAR_JERK 50.0000,EXAX_IGN 0}
DECL E6POS XPD={X 496.200287,Y 374.316742,Z 330.279724,A 43.3064499,B -1.60716689,C 179.054642,S 2,T 3,E1 0.0,E2 0.0,E3 0.0,E4 0.0,E5 0.0,E6 0.0}
DECL FDAT FPD={TOOL_NO 1,BASE_NO 0,IPO_FRAME #BASE,POINT2[] " ",TQ_STATE FALSE}
DECL LDAT LCPDAT12={VEL 2.00000,ACC 100.000,APO_DIST 100.000,APO_FAC 50.0000,AXIS_VEL 100.000,AXIS_ACC 100.000,ORI_TYP #VAR,CIRC_TYP #BASE,JERK_FAC 50.0000,GEAR_JERK 50.0000,EXAX_IGN 0}
DECL E6POS XPDA={X 496.200287,Y 374.316742,Z 450.351959,A 43.3064499,B -1.60716689,C 179.054642,S 2,T 3,E1 0.0,E2 0.0,E3 0.0,E4 0.0,E5 0.0,E6 0.0}
DECL FDAT FPDA={TOOL_NO 1,BASE_NO 0,IPO_FRAME #BASE,POINT2[] " ",TQ_STATE FALSE}
DECL LDAT LCPDAT13={VEL 2.00000,ACC 100.000,APO_DIST 100.000,APO_FAC 50.0000,AXIS_VEL 100.000,AXIS_ACC 100.000,ORI_TYP #VAR,CIRC_TYP #BASE,JERK_FAC 50.0000,GEAR_JERK 50.0000,EXAX_IGN 0}
DECL LDAT LCPDAT14={VEL 2.00000,ACC 100.000,APO_DIST 100.000,APO_FAC 50.0000,AXIS_VEL 100.000,AXIS_ACC 100.000,ORI_TYP #VAR,CIRC_TYP #BASE,JERK_FAC 50.0000,GEAR_JERK 50.0000,EXAX_IGN 0}
DECL E6POS XPDP={X 505.181946,Y 75.1278763,Z 340.542236,A 43.3075371,B -1.64983118,C 179.024796,S 2,T 11,E1 0.0,E2 0.0,E3 0.0,E4 0.0,E5 0.0,E6 0.0}
DECL FDAT Fpdp={TOOL_NO 1,BASE_NO 0,IPO_FRAME #BASE,POINT2[] " ",TQ_STATE FALSE}
DECL E6POS XPDPA={X 505.181946,Y 75.1278763,Z 469.675323,A 43.3075371,B -1.64983118,C 179.024796,S 2,T 11,E1 0.0,E2 0.0,E3 0.0,E4 0.0,E5 0.0,E6 0.0}
DECL FDAT Fpdpa={TOOL_NO 1,BASE_NO 0,IPO_FRAME #BASE,POINT2[] " ",TQ_STATE FALSE}
DECL LDAT LCPDAT15={VEL 2.00000,ACC 100.000,APO_DIST 100.000,APO_FAC 50.0000,AXIS_VEL 100.000,AXIS_ACC 100.000,ORI_TYP #VAR,CIRC_TYP #BASE,JERK_FAC 50.0000,GEAR_JERK 50.0000,EXAX_IGN 0}
DECL E6POS XCENTROVENTS={X 222.016174,Y -373.681549,Z 503.684784,A -46.3701553,B 0.222000524,C 179.228622,S 2,T 2,E1 0.0,E2 0.0,E3 0.0,E4 0.0,E5 0.0,E6 0.0}
DECL FDAT Fcentrovents={TOOL_NO 1,BASE_NO 0,IPO_FRAME #BASE,POINT2[] " ",TQ_STATE FALSE}
DECL PDAT PPDAT8={VEL 100.000,ACC 100.000,APO_DIST 100.000,APO_MODE #CDIS,GEAR_JERK 50.0000,EXAX_IGN 0}
DECL E6POS XVENT1={X 442.304138,Y -397.379,Z 155.349716,A -46.3701591,B 0.221998900,C 179.228592,S 2,T 2,E1 0.0,E2 0.0,E3 0.0,E4 0.0,E5 0.0,E6 0.0}
DECL FDAT Fvent1={TOOL_NO 1,BASE_NO 0,IPO_FRAME #BASE,POINT2[] " ",TQ_STATE FALSE}
DECL PDAT PPDAT9={VEL 100.000,ACC 100.000,APO_DIST 100.000,APO_MODE #CDIS,GEAR_JERK 50.0000,EXAX_IGN 0}
DECL E6POS XVENTA={X 442.304138,Y -397.379,Z 395.456726,A -46.3701591,B 0.221998885,C 179.228592,S 2,T 2,E1 0.0,E2 0.0,E3 0.0,E4 0.0,E5 0.0,E6 0.0}
DECL FDAT FventA={TOOL_NO 1,BASE_NO 0,IPO_FRAME #BASE,POINT2[] " ",TQ_STATE FALSE}
DECL LDAT LCPDAT16={VEL 2.00000,ACC 100.000,APO_DIST 100.000,APO_FAC 50.0000,AXIS_VEL 100.000,AXIS_ACC 100.000,ORI_TYP #VAR,CIRC_TYP #BASE,JERK_FAC 50.0000,GEAR_JERK 50.0000,EXAX_IGN 0}
DECL LDAT LCPDAT17={VEL 2.00000,ACC 100.000,APO_DIST 100.000,APO_FAC 50.0000,AXIS_VEL 100.000,AXIS_ACC 100.000,ORI_TYP #VAR,CIRC_TYP #BASE,JERK_FAC 50.0000,GEAR_JERK 50.0000,EXAX_IGN 0}
DECL E6POS XVENTA2={X 415.256256,Y -14.7377806,Z 509.505,A -46.3701591,B 0.221998855,C 179.228592,S 2,T 2,E1 0.0,E2 0.0,E3 0.0,E4 0.0,E5 0.0,E6 0.0}
DECL FDAT FventA2={TOOL_NO 1,BASE_NO 0,IPO_FRAME #BASE,POINT2[] " ",TQ_STATE FALSE}
DECL PDAT PPDAT10={VEL 100.000,ACC 100.000,APO_DIST 100.000,APO_MODE #CDIS,GEAR_JERK 50.0000,EXAX_IGN 0}
DECL E6POS XVENT1P={X 499.485138,Y -8.99362,Z 244.693527,A -44.9232407,B -0.888244927,C -179.702423,S 2,T 3,E1 0.0,E2 0.0,E3 0.0,E4 0.0,E5 0.0,E6 0.0}
DECL FDAT Fvent1P={TOOL_NO 1,BASE_NO 0,IPO_FRAME #BASE,POINT2[] " ",TQ_STATE FALSE}
DECL LDAT LCPDAT18={VEL 2.00000,ACC 100.000,APO_DIST 100.000,APO_FAC 50.0000,AXIS_VEL 100.000,AXIS_ACC 100.000,ORI_TYP #VAR,CIRC_TYP #BASE,JERK_FAC 50.0000,GEAR_JERK 50.0000,EXAX_IGN 0}
DECL E6POS XVENT1AA={X 499.485138,Y -8.99362,Z 532.041199,A -44.9232407,B -0.888244927,C -179.702423,S 2,T 3,E1 0.0,E2 0.0,E3 0.0,E4 0.0,E5 0.0,E6 0.0}
DECL FDAT Fvent1AA={TOOL_NO 1,BASE_NO 0,IPO_FRAME #BASE,POINT2[] " ",TQ_STATE FALSE}
DECL LDAT LCPDAT19={VEL 2.00000,ACC 100.000,APO_DIST 100.000,APO_FAC 50.0000,AXIS_VEL 100.000,AXIS_ACC 100.000,ORI_TYP #VAR,CIRC_TYP #BASE,JERK_FAC 50.0000,GEAR_JERK 50.0000,EXAX_IGN 0}
DECL E6POS Xvent1P_1={X 499.485138,Y -8.99362,Z 244.693527,A -44.9232407,B -0.888244927,C -179.702423,S 2,T 3,E1 0.0,E2 0.0,E3 0.0,E4 0.0,E5 0.0,E6 0.0}
DECL FDAT Fvent1P_1={TOOL_NO 1,BASE_NO 0,IPO_FRAME #BASE,POINT2[] " ",TQ_STATE FALSE}
DECL LDAT LCPDAT38={VEL 2.00000,ACC 100.000,APO_DIST 100.000,APO_FAC 50.0000,AXIS_VEL 100.000,AXIS_ACC 100.000,ORI_TYP #VAR,CIRC_TYP #BASE,JERK_FAC 50.0000,GEAR_JERK 50.0000,EXAX_IGN 0}
DECL E6POS Xvent1AA_1={X 499.485138,Y -8.99362,Z 532.041199,A -44.9232407,B -0.888244927,C -179.702423,S 2,T 3,E1 0.0,E2 0.0,E3 0.0,E4 0.0,E5 0.0,E6 0.0}
DECL FDAT Fvent1AA_1={TOOL_NO 1,BASE_NO 0,IPO_FRAME #BASE,POINT2[] " ",TQ_STATE FALSE}
DECL LDAT LCPDAT37={VEL 2.00000,ACC 100.000,APO_DIST 100.000,APO_FAC 50.0000,AXIS_VEL 100.000,AXIS_ACC 100.000,ORI_TYP #VAR,CIRC_TYP #BASE,JERK_FAC 50.0000,GEAR_JERK 50.0000,EXAX_IGN 0}
DECL E6POS Xvent2={X 442.304138,Y -397.379,Z 155.349716,A -46.3701591,B 0.221998900,C 179.228592,S 2,T 2,E1 0.0,E2 0.0,E3 0.0,E4 0.0,E5 0.0,E6 0.0}
DECL FDAT Fvent2={TOOL_NO 1,BASE_NO 0,IPO_FRAME #BASE,POINT2[] " ",TQ_STATE FALSE}
DECL LDAT LCPDAT36={VEL 2.00000,ACC 100.000,APO_DIST 100.000,APO_FAC 50.0000,AXIS_VEL 100.000,AXIS_ACC 100.000,ORI_TYP #VAR,CIRC_TYP #BASE,JERK_FAC 50.0000,GEAR_JERK 50.0000,EXAX_IGN 0}
DECL E6POS XventA_1={X 442.304138,Y -397.379,Z 395.456726,A -46.3701591,B 0.221998885,C 179.228592,S 2,T 2,E1 0.0,E2 0.0,E3 0.0,E4 0.0,E5 0.0,E6 0.0}
DECL FDAT FventA_1={TOOL_NO 1,BASE_NO 0,IPO_FRAME #BASE,POINT2[] " ",TQ_STATE FALSE}
DECL LDAT LCPDAT35={VEL 2.00000,ACC 100.000,APO_DIST 100.000,APO_FAC 50.0000,AXIS_VEL 100.000,AXIS_ACC 100.000,ORI_TYP #VAR,CIRC_TYP #BASE,JERK_FAC 50.0000,GEAR_JERK 50.0000,EXAX_IGN 0}
DECL E6POS XventA3={X 415.256256,Y -14.7377806,Z 509.505,A -46.3701591,B 0.221998855,C 179.228592,S 2,T 2,E1 0.0,E2 0.0,E3 0.0,E4 0.0,E5 0.0,E6 0.0}
DECL FDAT FventA3={TOOL_NO 1,BASE_NO 0,IPO_FRAME #BASE,POINT2[] " ",TQ_STATE FALSE}
DECL PDAT PPDAT14={VEL 100.000,ACC 100.000,APO_DIST 100.000,APO_MODE #CDIS,GEAR_JERK 50.0000,EXAX_IGN 0}
DECL E6POS Xpdp_1={X 505.181946,Y 75.1278763,Z 340.542236,A 43.3075371,B -1.64983118,C 179.024796,S 2,T 11,E1 0.0,E2 0.0,E3 0.0,E4 0.0,E5 0.0,E6 0.0}
DECL FDAT Fpdp_1={TOOL_NO 1,BASE_NO 0,IPO_FRAME #BASE,POINT2[] " ",TQ_STATE FALSE}
DECL LDAT LCPDAT34={VEL 2.00000,ACC 100.000,APO_DIST 100.000,APO_FAC 50.0000,AXIS_VEL 100.000,AXIS_ACC 100.000,ORI_TYP #VAR,CIRC_TYP #BASE,JERK_FAC 50.0000,GEAR_JERK 50.0000,EXAX_IGN 0}
DECL E6POS Xpdpa_1={X 505.181946,Y 75.1278763,Z 469.675323,A 43.3075371,B -1.64983118,C 179.024796,S 2,T 11,E1 0.0,E2 0.0,E3 0.0,E4 0.0,E5 0.0,E6 0.0}
DECL FDAT Fpdpa_1={TOOL_NO 1,BASE_NO 0,IPO_FRAME #BASE,POINT2[] " ",TQ_STATE FALSE}
DECL LDAT LCPDAT33={VEL 2.00000,ACC 100.000,APO_DIST 100.000,APO_FAC 50.0000,AXIS_VEL 100.000,AXIS_ACC 100.000,ORI_TYP #VAR,CIRC_TYP #BASE,JERK_FAC 50.0000,GEAR_JERK 50.0000,EXAX_IGN 0}
DECL E6POS XPD_1={X 496.200287,Y 374.316742,Z 330.279724,A 43.3064499,B -1.60716689,C 179.054642,S 2,T 3,E1 0.0,E2 0.0,E3 0.0,E4 0.0,E5 0.0,E6 0.0}
DECL FDAT FPD_1={TOOL_NO 1,BASE_NO 0,IPO_FRAME #BASE,POINT2[] " ",TQ_STATE FALSE}
DECL LDAT LCPDAT32={VEL 2.00000,ACC 100.000,APO_DIST 100.000,APO_FAC 50.0000,AXIS_VEL 100.000,AXIS_ACC 100.000,ORI_TYP #VAR,CIRC_TYP #BASE,JERK_FAC 50.0000,GEAR_JERK 50.0000,EXAX_IGN 0}
DECL E6POS XPDA_1={X 496.200287,Y 374.316742,Z 450.351959,A 43.3064499,B -1.60716689,C 179.054642,S 2,T 3,E1 0.0,E2 0.0,E3 0.0,E4 0.0,E5 0.0,E6 0.0}
DECL FDAT FPDA_1={TOOL_NO 1,BASE_NO 0,IPO_FRAME #BASE,POINT2[] " ",TQ_STATE FALSE}
DECL LDAT LCPDAT31={VEL 2.00000,ACC 100.000,APO_DIST 100.000,APO_FAC 50.0000,AXIS_VEL 100.000,AXIS_ACC 100.000,ORI_TYP #VAR,CIRC_TYP #BASE,JERK_FAC 50.0000,GEAR_JERK 50.0000,EXAX_IGN 0}
DECL E6POS Xpip_1={X 503.498657,Y -68.2245560,Z 339.513977,A 43.3322525,B -1.62203932,C 179.037308,S 2,T 10,E1 0.0,E2 0.0,E3 0.0,E4 0.0,E5 0.0,E6 0.0}
DECL FDAT Fpip_1={TOOL_NO 1,BASE_NO 0,IPO_FRAME #BASE,POINT2[] " ",TQ_STATE FALSE}
DECL LDAT LCPDAT30={VEL 2.00000,ACC 100.000,APO_DIST 100.000,APO_FAC 50.0000,AXIS_VEL 100.000,AXIS_ACC 100.000,ORI_TYP #VAR,CIRC_TYP #BASE,JERK_FAC 50.0000,GEAR_JERK 50.0000,EXAX_IGN 0}
DECL E6POS Xpipa_1={X 503.395630,Y -68.2099609,Z 442.073,A 43.3303375,B -1.60676658,C 179.056412,S 2,T 10,E1 0.0,E2 0.0,E3 0.0,E4 0.0,E5 0.0,E6 0.0}
DECL FDAT Fpipa_1={TOOL_NO 1,BASE_NO 0,IPO_FRAME #BASE,POINT2[] " ",TQ_STATE FALSE}
DECL LDAT LCPDAT29={VEL 2.00000,ACC 100.000,APO_DIST 100.000,APO_FAC 50.0000,AXIS_VEL 100.000,AXIS_ACC 100.000,ORI_TYP #VAR,CIRC_TYP #BASE,JERK_FAC 50.0000,GEAR_JERK 50.0000,EXAX_IGN 0}
DECL E6POS XPI_1={X 488.794952,Y 263.522217,Z 330.558746,A 38.9071503,B -1.58586621,C 179.083191,S 2,T 3,E1 0.0,E2 0.0,E3 0.0,E4 0.0,E5 0.0,E6 0.0}
DECL FDAT FPI_1={TOOL_NO 1,BASE_NO 0,IPO_FRAME #BASE,POINT2[] " ",TQ_STATE FALSE}
DECL LDAT LCPDAT28={VEL 2.00000,ACC 100.000,APO_DIST 100.000,APO_FAC 50.0000,AXIS_VEL 100.000,AXIS_ACC 100.000,ORI_TYP #VAR,CIRC_TYP #BASE,JERK_FAC 50.0000,GEAR_JERK 50.0000,EXAX_IGN 0}
DECL E6POS XPIA_1={X 488.794952,Y 263.522217,Z 467.844391,A 38.9071503,B -1.58586633,C 179.083191,S 2,T 3,E1 0.0,E2 0.0,E3 0.0,E4 0.0,E5 0.0,E6 0.0}
DECL FDAT FPIA_1={TOOL_NO 1,BASE_NO 0,IPO_FRAME #BASE,POINT2[] " ",TQ_STATE FALSE}
DECL LDAT LCPDAT27={VEL 2.00000,ACC 100.000,APO_DIST 100.000,APO_FAC 50.0000,AXIS_VEL 100.000,AXIS_ACC 100.000,ORI_TYP #VAR,CIRC_TYP #BASE,JERK_FAC 50.0000,GEAR_JERK 50.0000,EXAX_IGN 0}
DECL E6POS XcodoDP_1={X 495.551361,Y 75.4896164,Z 104.322121,A 42.5106506,B -1.61344421,C 179.062820,S 2,T 11,E1 0.0,E2 0.0,E3 0.0,E4 0.0,E5 0.0,E6 0.0}
DECL FDAT FcodoDP_1={TOOL_NO 1,BASE_NO 0,IPO_FRAME #BASE,POINT2[] " ",TQ_STATE FALSE}
DECL LDAT LCPDAT26={VEL 2.00000,ACC 100.000,APO_DIST 100.000,APO_FAC 50.0000,AXIS_VEL 100.000,AXIS_ACC 100.000,ORI_TYP #VAR,CIRC_TYP #BASE,JERK_FAC 50.0000,GEAR_JERK 50.0000,EXAX_IGN 0}
DECL E6POS XcodoDPA_1={X 495.551361,Y 75.4896164,Z 295.991516,A 42.5106506,B -1.61344421,C 179.062820,S 2,T 11,E1 0.0,E2 0.0,E3 0.0,E4 0.0,E5 0.0,E6 0.0}
DECL FDAT FcodoDPA_1={TOOL_NO 1,BASE_NO 0,IPO_FRAME #BASE,POINT2[] " ",TQ_STATE FALSE}
DECL PDAT PPDAT13={VEL 100.000,ACC 100.000,APO_DIST 100.000,APO_MODE #CDIS,GEAR_JERK 50.0000,EXAX_IGN 0}
DECL E6POS XcodoD_1={X 120.584869,Y 330.035919,Z 251.804016,A -5.40004730,B 17.7066059,C -156.192,S 2,T 11,E1 0.0,E2 0.0,E3 0.0,E4 0.0,E5 0.0,E6 0.0}
DECL FDAT FcodoD_1={TOOL_NO 1,BASE_NO 0,IPO_FRAME #BASE,POINT2[] " ",TQ_STATE FALSE}
DECL LDAT LCPDAT25={VEL 2.00000,ACC 100.000,APO_DIST 100.000,APO_FAC 50.0000,AXIS_VEL 100.000,AXIS_ACC 100.000,ORI_TYP #VAR,CIRC_TYP #BASE,JERK_FAC 50.0000,GEAR_JERK 50.0000,EXAX_IGN 0}
DECL E6POS XcodoD3={X 120.584869,Y 330.035919,Z 422.057,A -5.40004730,B 17.7066059,C -156.192,S 2,T 11,E1 0.0,E2 0.0,E3 0.0,E4 0.0,E5 0.0,E6 0.0}
DECL FDAT FcodoD3={TOOL_NO 1,BASE_NO 0,IPO_FRAME #BASE,POINT2[] " ",TQ_STATE FALSE}
DECL PDAT PPDAT12={VEL 100.000,ACC 100.000,APO_DIST 100.000,APO_MODE #CDIS,GEAR_JERK 50.0000,EXAX_IGN 0}
DECL E6POS XcodoIP_1={X 495.259338,Y -72.1194916,Z 105.335014,A 42.5121155,B -1.58614099,C 179.082733,S 2,T 10,E1 0.0,E2 0.0,E3 0.0,E4 0.0,E5 0.0,E6 0.0}
DECL FDAT FcodoIP_1={TOOL_NO 1,BASE_NO 0,IPO_FRAME #BASE,POINT2[] " ",TQ_STATE FALSE}
DECL LDAT LCPDAT24={VEL 2.00000,ACC 100.000,APO_DIST 100.000,APO_FAC 50.0000,AXIS_VEL 100.000,AXIS_ACC 100.000,ORI_TYP #VAR,CIRC_TYP #BASE,JERK_FAC 50.0000,GEAR_JERK 50.0000,EXAX_IGN 0}
DECL E6POS XcodoIPA_1={X 495.277374,Y -72.1219254,Z 305.970398,A 42.5108,B -1.58776,C 179.080200,S 2,T 10,E1 0.0,E2 0.0,E3 0.0,E4 0.0,E5 0.0,E6 0.0}
DECL FDAT FcodoIPA_1={TOOL_NO 1,BASE_NO 0,IPO_FRAME #BASE,POINT2[] " ",TQ_STATE FALSE}
DECL LDAT LCPDAT23={VEL 2.00000,ACC 100.000,APO_DIST 100.000,APO_FAC 50.0000,AXIS_VEL 100.000,AXIS_ACC 100.000,ORI_TYP #VAR,CIRC_TYP #BASE,JERK_FAC 50.0000,GEAR_JERK 50.0000,EXAX_IGN 0}
DECL E6POS XcodoIB_1={X 169.580139,Y 270.518555,Z 98.2024536,A -5.40927553,B 17.7038708,C -156.222351,S 2,T 11,E1 0.0,E2 0.0,E3 0.0,E4 0.0,E5 0.0,E6 0.0}
DECL FDAT FcodoIB_1={TOOL_NO 1,BASE_NO 0,IPO_FRAME #BASE,POINT2[] " ",TQ_STATE FALSE}
DECL LDAT LCPDAT22={VEL 2.00000,ACC 100.000,APO_DIST 100.000,APO_FAC 50.0000,AXIS_VEL 100.000,AXIS_ACC 100.000,ORI_TYP #VAR,CIRC_TYP #BASE,JERK_FAC 50.0000,GEAR_JERK 50.0000,EXAX_IGN 0}
DECL E6POS XcodoIB5={X 169.370163,Y 288.233887,Z 215.088318,A -9.98564243,B -1.58595812,C 179.083130,S 2,T 3,E1 0.0,E2 0.0,E3 0.0,E4 0.0,E5 0.0,E6 0.0}
DECL FDAT FcodoIB5={TOOL_NO 1,BASE_NO 0,IPO_FRAME #BASE,POINT2[] " ",TQ_STATE FALSE}
DECL LDAT LCPDAT21={VEL 2.00000,ACC 100.000,APO_DIST 100.000,APO_FAC 50.0000,AXIS_VEL 100.000,AXIS_ACC 100.000,ORI_TYP #VAR,CIRC_TYP #BASE,JERK_FAC 50.0000,GEAR_JERK 50.0000,EXAX_IGN 0}
DECL E6POS XcodoIB4={X 169.372009,Y 288.237305,Z 503.685242,A -9.98564529,B -1.58597386,C 179.083130,S 2,T 3,E1 0.0,E2 0.0,E3 0.0,E4 0.0,E5 0.0,E6 0.0}
DECL FDAT FcodoIB4={TOOL_NO 1,BASE_NO 0,IPO_FRAME #BASE,POINT2[] " ",TQ_STATE FALSE}
DECL LDAT LCPDAT20={VEL 2.00000,ACC 100.000,APO_DIST 100.000,APO_FAC 50.0000,AXIS_VEL 100.000,AXIS_ACC 100.000,ORI_TYP #VAR,CIRC_TYP #BASE,JERK_FAC 50.0000,GEAR_JERK 50.0000,EXAX_IGN 0}
DECL E6POS Xcentro_1={X 222.017685,Y 1.93147576,Z 503.686340,A 38.9071503,B -1.58586597,C 179.083191,S 2,T 10,E1 0.0,E2 0.0,E3 0.0,E4 0.0,E5 0.0,E6 0.0}
DECL FDAT Fcentro_1={TOOL_NO 1,BASE_NO 0,IPO_FRAME #BASE,POINT2[] " ",TQ_STATE FALSE}
DECL PDAT PPDAT11={VEL 100.000,ACC 100.000,APO_DIST 100.000,APO_MODE #CDIS,GEAR_JERK 50.0000,EXAX_IGN 0}
DECL E6POS Xcentro_2={X 222.017685,Y 1.93147576,Z 503.686340,A 38.9071503,B -1.58586597,C 179.083191,S 2,T 10,E1 0.0,E2 0.0,E3 0.0,E4 0.0,E5 0.0,E6 0.0}
DECL FDAT Fcentro_2={TOOL_NO 1,BASE_NO 0,IPO_FRAME #BASE,POINT2[] " ",TQ_STATE FALSE}
DECL PDAT PPDAT15={VEL 100.000,ACC 100.000,APO_DIST 100.000,APO_MODE #CDIS,GEAR_JERK 50.0000,EXAX_IGN 0}
DECL E6POS Xcentro_3={X 222.017685,Y 1.93147576,Z 503.686340,A 38.9071503,B -1.58586597,C 179.083191,S 2,T 10,E1 0.0,E2 0.0,E3 0.0,E4 0.0,E5 0.0,E6 0.0}
DECL FDAT Fcentro_3={TOOL_NO 1,BASE_NO 0,IPO_FRAME #BASE,POINT2[] " ",TQ_STATE FALSE}
DECL PDAT PPDAT16={VEL 100.000,ACC 100.000,APO_DIST 100.000,APO_MODE #CDIS,GEAR_JERK 50.0000,EXAX_IGN 0}
DECL E6POS XVENT3AA={X 264.549,Y -226.508316,Z 557.449402,A -139.096802,B -19.1079426,C -157.486145,S 2,T 2,E1 0.0,E2 0.0,E3 0.0,E4 0.0,E5 0.0,E6 0.0}
DECL FDAT Fvent3aa={TOOL_NO 1,BASE_NO 0,IPO_FRAME #BASE,POINT2[] " ",TQ_STATE FALSE}
DECL PDAT PPDAT17={VEL 100.000,ACC 100.000,APO_DIST 100.000,APO_MODE #CDIS,GEAR_JERK 50.0000,EXAX_IGN 0}
DECL E6POS XVENT4AA={X 264.553955,Y -220.491226,Z 198.112228,A -139.098389,B -19.1098919,C -157.483841,S 2,T 2,E1 0.0,E2 0.0,E3 0.0,E4 0.0,E5 0.0,E6 0.0}
DECL FDAT Fvent4aa={TOOL_NO 1,BASE_NO 0,IPO_FRAME #BASE,POINT2[] " ",TQ_STATE FALSE}
DECL LDAT LCPDAT39={VEL 2.00000,ACC 100.000,APO_DIST 100.000,APO_FAC 50.0000,AXIS_VEL 100.000,AXIS_ACC 100.000,ORI_TYP #VAR,CIRC_TYP #BASE,JERK_FAC 50.0000,GEAR_JERK 50.0000,EXAX_IGN 0}
DECL E6POS XVENT5AA={X 264.555847,Y -253.658203,Z 144.983124,A -139.099091,B -19.1109238,C -157.482803,S 2,T 34,E1 0.0,E2 0.0,E3 0.0,E4 0.0,E5 0.0,E6 0.0}
DECL FDAT Fvent5aa={TOOL_NO 1,BASE_NO 0,IPO_FRAME #BASE,POINT2[] " ",TQ_STATE FALSE}
DECL LDAT LCPDAT40={VEL 2.00000,ACC 100.000,APO_DIST 100.000,APO_FAC 50.0000,AXIS_VEL 100.000,AXIS_ACC 100.000,ORI_TYP #VAR,CIRC_TYP #BASE,JERK_FAC 50.0000,GEAR_JERK 50.0000,EXAX_IGN 0}
DECL E6POS XVENT6AA={X 264.557220,Y -218.268707,Z 210.296631,A -139.099686,B -19.1118259,C -157.481949,S 2,T 2,E1 0.0,E2 0.0,E3 0.0,E4 0.0,E5 0.0,E6 0.0}
DECL FDAT Fvent6aa={TOOL_NO 1,BASE_NO 0,IPO_FRAME #BASE,POINT2[] " ",TQ_STATE FALSE}
DECL LDAT LCPDAT41={VEL 2.00000,ACC 100.000,APO_DIST 100.000,APO_FAC 50.0000,AXIS_VEL 100.000,AXIS_ACC 100.000,ORI_TYP #VAR,CIRC_TYP #BASE,JERK_FAC 50.0000,GEAR_JERK 50.0000,EXAX_IGN 0}
DECL E6POS XVENT7AA={X 264.557251,Y -184.106232,Z 273.886200,A -139.099701,B -19.1118355,C -157.481934,S 2,T 2,E1 0.0,E2 0.0,E3 0.0,E4 0.0,E5 0.0,E6 0.0}
DECL FDAT Fvent7aa={TOOL_NO 1,BASE_NO 0,IPO_FRAME #BASE,POINT2[] " ",TQ_STATE FALSE}
DECL LDAT LCPDAT42={VEL 2.00000,ACC 100.000,APO_DIST 100.000,APO_FAC 50.0000,AXIS_VEL 100.000,AXIS_ACC 100.000,ORI_TYP #VAR,CIRC_TYP #BASE,JERK_FAC 50.0000,GEAR_JERK 50.0000,EXAX_IGN 0}
DECL E6POS XVENT8AA={X 264.461761,Y 5.13799143,Z 584.457214,A 131.982437,B 1.28507471,C -178.538467,S 2,T 35,E1 0.0,E2 0.0,E3 0.0,E4 0.0,E5 0.0,E6 0.0}
DECL FDAT Fvent8aa={TOOL_NO 1,BASE_NO 0,IPO_FRAME #BASE,POINT2[] " ",TQ_STATE FALSE}
DECL PDAT PPDAT18={VEL 100.000,ACC 100.000,APO_DIST 100.000,APO_MODE #CDIS,GEAR_JERK 50.0000,EXAX_IGN 0}
DECL E6POS Xcentro_4={X 222.017685,Y 1.93147576,Z 503.686340,A 38.9071503,B -1.58586597,C 179.083191,S 2,T 10,E1 0.0,E2 0.0,E3 0.0,E4 0.0,E5 0.0,E6 0.0}
DECL FDAT Fcentro_4={TOOL_NO 1,BASE_NO 0,IPO_FRAME #BASE,POINT2[] " ",TQ_STATE FALSE}
DECL PDAT PPDAT19={VEL 100.000,ACC 100.000,APO_DIST 100.000,APO_MODE #CDIS,GEAR_JERK 50.0000,EXAX_IGN 0}
DECL E6POS XPIP2={X 503.418396,Y -75.2706299,Z 419.404022,A 43.3307610,B -1.61014235,C 179.052185,S 2,T 10,E1 0.0,E2 0.0,E3 0.0,E4 0.0,E5 0.0,E6 0.0}
DECL FDAT Fpip2={TOOL_NO 1,BASE_NO 0,IPO_FRAME #BASE,POINT2[] " ",TQ_STATE FALSE}
DECL LDAT LCPDAT43={VEL 2.00000,ACC 100.000,APO_DIST 100.000,APO_FAC 50.0000,AXIS_VEL 100.000,AXIS_ACC 100.000,ORI_TYP #VAR,CIRC_TYP #BASE,JERK_FAC 50.0000,GEAR_JERK 50.0000,EXAX_IGN 0}
DECL E6POS Xcentro_5={X 222.017685,Y 1.93147576,Z 503.686340,A 38.9071503,B -1.58586597,C 179.083191,S 2,T 10,E1 0.0,E2 0.0,E3 0.0,E4 0.0,E5 0.0,E6 0.0}
DECL FDAT Fcentro_5={TOOL_NO 1,BASE_NO 0,IPO_FRAME #BASE,POINT2[] " ",TQ_STATE FALSE}
DECL PDAT PPDAT20={VEL 100.000,ACC 100.000,APO_DIST 100.000,APO_MODE #CDIS,GEAR_JERK 50.0000,EXAX_IGN 0}
DECL E6POS XIB2={X 171.637909,Y 270.518555,Z 94.8026123,A -5.17180,B 20.3039608,C -155.420685,S 2,T 11,E1 0.0,E2 0.0,E3 0.0,E4 0.0,E5 0.0,E6 0.0}
DECL FDAT FIB2={TOOL_NO 1,BASE_NO 0,IPO_FRAME #BASE,POINT2[] " ",TQ_STATE FALSE}
DECL LDAT LCPDAT44={VEL 2.00000,ACC 100.000,APO_DIST 100.000,APO_FAC 50.0000,AXIS_VEL 100.000,AXIS_ACC 100.000,ORI_TYP #VAR,CIRC_TYP #BASE,JERK_FAC 50.0000,GEAR_JERK 50.0000,EXAX_IGN 0}
DECL E6POS XIB3={X 172.239731,Y 269.638824,Z 111.731445,A -6.09838581,B 20.0551949,C -158.106277,S 2,T 11,E1 0.0,E2 0.0,E3 0.0,E4 0.0,E5 0.0,E6 0.0}
DECL FDAT FIB3={TOOL_NO 1,BASE_NO 0,IPO_FRAME #BASE,POINT2[] " ",TQ_STATE FALSE}
DECL LDAT LCPDAT45={VEL 2.00000,ACC 100.000,APO_DIST 100.000,APO_FAC 50.0000,AXIS_VEL 100.000,AXIS_ACC 100.000,ORI_TYP #VAR,CIRC_TYP #BASE,JERK_FAC 50.0000,GEAR_JERK 50.0000,EXAX_IGN 0}
DECL E6POS XIP2={X 493.945343,Y -71.5176544,Z 120.988960,A 42.5177116,B -1.73602641,C 178.891678,S 2,T 10,E1 0.0,E2 0.0,E3 0.0,E4 0.0,E5 0.0,E6 0.0}
DECL FDAT FIP2={TOOL_NO 1,BASE_NO 0,IPO_FRAME #BASE,POINT2[] " ",TQ_STATE FALSE}
DECL LDAT LCPDAT46={VEL 2.00000,ACC 100.000,APO_DIST 100.000,APO_FAC 50.0000,AXIS_VEL 100.000,AXIS_ACC 100.000,ORI_TYP #VAR,CIRC_TYP #BASE,JERK_FAC 50.0000,GEAR_JERK 50.0000,EXAX_IGN 0}
DECL E6POS XIP3={X 492.207214,Y -71.4600372,Z 271.568909,A 42.5177116,B -1.73602641,C 178.891678,S 2,T 10,E1 0.0,E2 0.0,E3 0.0,E4 0.0,E5 0.0,E6 0.0}
DECL FDAT FIP3={TOOL_NO 1,BASE_NO 0,IPO_FRAME #BASE,POINT2[] " ",TQ_STATE FALSE}
DECL LDAT LCPDAT47={VEL 2.00000,ACC 100.000,APO_DIST 100.000,APO_FAC 50.0000,AXIS_VEL 100.000,AXIS_ACC 100.000,ORI_TYP #VAR,CIRC_TYP #BASE,JERK_FAC 50.0000,GEAR_JERK 50.0000,EXAX_IGN 0}
DECL LDAT LCPDAT48={VEL 2.00000,ACC 100.000,APO_DIST 100.000,APO_FAC 50.0000,AXIS_VEL 100.000,AXIS_ACC 100.000,ORI_TYP #VAR,CIRC_TYP #BASE,JERK_FAC 50.0000,GEAR_JERK 50.0000,EXAX_IGN 0}
DECL E6POS XCODOD4={X 124.531929,Y 329.923431,Z 264.745789,A -5.13479567,B 18.8223400,C -158.743607,S 2,T 11,E1 0.0,E2 0.0,E3 0.0,E4 0.0,E5 0.0,E6 0.0}
DECL FDAT FcodoD4={TOOL_NO 1,BASE_NO 0,IPO_FRAME #BASE,POINT2[] " ",TQ_STATE FALSE}
DECL PDAT PPDAT21={VEL 100.000,ACC 100.000,APO_DIST 100.000,APO_MODE #CDIS,GEAR_JERK 50.0000,EXAX_IGN 0}
DECL E6POS XCODOD5={X 495.551361,Y 76.0944138,Z 116.386284,A 42.5106506,B -1.61344540,C 179.062820,S 2,T 11,E1 0.0,E2 0.0,E3 0.0,E4 0.0,E5 0.0,E6 0.0}
DECL FDAT FcodoD5={TOOL_NO 1,BASE_NO 0,IPO_FRAME #BASE,POINT2[] " ",TQ_STATE FALSE}
DECL LDAT LCPDAT49={VEL 2.00000,ACC 100.000,APO_DIST 100.000,APO_FAC 50.0000,AXIS_VEL 100.000,AXIS_ACC 100.000,ORI_TYP #VAR,CIRC_TYP #BASE,JERK_FAC 50.0000,GEAR_JERK 50.0000,EXAX_IGN 0}
DECL E6POS XCODOD6={X 495.554962,Y 76.0949554,Z 319.206970,A 42.5106506,B -1.61344540,C 179.062820,S 2,T 11,E1 0.0,E2 0.0,E3 0.0,E4 0.0,E5 0.0,E6 0.0}
DECL FDAT FcodoD6={TOOL_NO 1,BASE_NO 0,IPO_FRAME #BASE,POINT2[] " ",TQ_STATE FALSE}
DECL LDAT LCPDAT50={VEL 2.00000,ACC 100.000,APO_DIST 100.000,APO_FAC 50.0000,AXIS_VEL 100.000,AXIS_ACC 100.000,ORI_TYP #VAR,CIRC_TYP #BASE,JERK_FAC 50.0000,GEAR_JERK 50.0000,EXAX_IGN 0}
DECL E6POS XRICK={X 494.507660,Y 75.6533051,Z 122.752953,A 45.7913361,B -3.70535922,C 177.634613,S 2,T 11,E1 0.0,E2 0.0,E3 0.0,E4 0.0,E5 0.0,E6 0.0}
DECL FDAT Frick={TOOL_NO 1,BASE_NO 0,IPO_FRAME #BASE,POINT2[] " ",TQ_STATE FALSE}
DECL LDAT LCPDAT51={VEL 2.00000,ACC 100.000,APO_DIST 100.000,APO_FAC 50.0000,AXIS_VEL 100.000,AXIS_ACC 100.000,ORI_TYP #VAR,CIRC_TYP #BASE,JERK_FAC 50.0000,GEAR_JERK 50.0000,EXAX_IGN 0}
DECL E6POS XRICK1={X 508.524597,Y -72.2787,Z 337.363647,A 43.3267899,B -1.63019383,C 179.026901,S 2,T 10,E1 0.0,E2 0.0,E3 0.0,E4 0.0,E5 0.0,E6 0.0}
DECL FDAT Frick1={TOOL_NO 1,BASE_NO 0,IPO_FRAME #BASE,POINT2[] " ",TQ_STATE FALSE}
DECL LDAT LCPDAT52={VEL 2.00000,ACC 100.000,APO_DIST 100.000,APO_FAC 50.0000,AXIS_VEL 100.000,AXIS_ACC 100.000,ORI_TYP #VAR,CIRC_TYP #BASE,JERK_FAC 50.0000,GEAR_JERK 50.0000,EXAX_IGN 0}
DECL E6POS XRICK2={X 494.467621,Y 75.6489792,Z 265.259155,A 45.7905807,B -3.69958639,C 177.638535,S 2,T 11,E1 0.0,E2 0.0,E3 0.0,E4 0.0,E5 0.0,E6 0.0}
DECL FDAT Frick2={TOOL_NO 1,BASE_NO 0,IPO_FRAME #BASE,POINT2[] " ",TQ_STATE FALSE}
DECL LDAT LCPDAT53={VEL 2.00000,ACC 100.000,APO_DIST 100.000,APO_FAC 50.0000,AXIS_VEL 100.000,AXIS_ACC 100.000,ORI_TYP #VAR,CIRC_TYP #BASE,JERK_FAC 50.0000,GEAR_JERK 50.0000,EXAX_IGN 0}
DECL E6POS XRICK3={X 510.790527,Y 70.2749252,Z 342.575317,A 44.8877525,B -0.653846085,C -179.850266,S 2,T 11,E1 0.0,E2 0.0,E3 0.0,E4 0.0,E5 0.0,E6 0.0}
DECL FDAT Frick3={TOOL_NO 1,BASE_NO 0,IPO_FRAME #BASE,POINT2[] " ",TQ_STATE FALSE}
DECL LDAT LCPDAT54={VEL 2.00000,ACC 100.000,APO_DIST 100.000,APO_FAC 50.0000,AXIS_VEL 100.000,AXIS_ACC 100.000,ORI_TYP #VAR,CIRC_TYP #BASE,JERK_FAC 50.0000,GEAR_JERK 50.0000,EXAX_IGN 0}
DECL E6POS XRICK4={X 510.798248,Y 70.2759705,Z 464.118958,A 44.8877525,B -0.653853238,C -179.850250,S 2,T 11,E1 0.0,E2 0.0,E3 0.0,E4 0.0,E5 0.0,E6 0.0}
DECL FDAT Frick4={TOOL_NO 1,BASE_NO 0,IPO_FRAME #BASE,POINT2[] " ",TQ_STATE FALSE}
DECL LDAT LCPDAT55={VEL 2.00000,ACC 100.000,APO_DIST 100.000,APO_FAC 50.0000,AXIS_VEL 100.000,AXIS_ACC 100.000,ORI_TYP #VAR,CIRC_TYP #BASE,JERK_FAC 50.0000,GEAR_JERK 50.0000,EXAX_IGN 0}
DECL E6POS XRICK5={X 510.465637,Y -75.1966705,Z 342.277863,A 43.6111870,B -0.562470794,C 179.257294,S 2,T 2,E1 0.0,E2 0.0,E3 0.0,E4 0.0,E5 0.0,E6 0.0}
DECL FDAT Frick5={TOOL_NO 1,BASE_NO 0,IPO_FRAME #BASE,POINT2[] " ",TQ_STATE FALSE}
DECL LDAT LCPDAT56={VEL 2.00000,ACC 100.000,APO_DIST 100.000,APO_FAC 50.0000,AXIS_VEL 100.000,AXIS_ACC 100.000,ORI_TYP #VAR,CIRC_TYP #BASE,JERK_FAC 50.0000,GEAR_JERK 50.0000,EXAX_IGN 0}
DECL E6POS XRICK6={X 510.444672,Y -75.1928940,Z 514.698914,A 43.6145935,B -0.547352850,C 179.277054,S 2,T 2,E1 0.0,E2 0.0,E3 0.0,E4 0.0,E5 0.0,E6 0.0}
DECL FDAT Frick6={TOOL_NO 1,BASE_NO 0,IPO_FRAME #BASE,POINT2[] " ",TQ_STATE FALSE}
DECL LDAT LCPDAT57={VEL 2.00000,ACC 100.000,APO_DIST 100.000,APO_FAC 50.0000,AXIS_VEL 100.000,AXIS_ACC 100.000,ORI_TYP #VAR,CIRC_TYP #BASE,JERK_FAC 50.0000,GEAR_JERK 50.0000,EXAX_IGN 0}
DECL E6POS XRICK7={X 500.839142,Y 7.79965878,Z 570.627441,A 132.153961,B 1.28462303,C -178.538376,S 2,T 35,E1 0.0,E2 0.0,E3 0.0,E4 0.0,E5 0.0,E6 0.0}
DECL FDAT Frick7={TOOL_NO 1,BASE_NO 0,IPO_FRAME #BASE,POINT2[] " ",TQ_STATE FALSE}
DECL LDAT LCPDAT58={VEL 2.00000,ACC 100.000,APO_DIST 100.000,APO_FAC 50.0000,AXIS_VEL 100.000,AXIS_ACC 100.000,ORI_TYP #VAR,CIRC_TYP #BASE,JERK_FAC 50.0000,GEAR_JERK 50.0000,EXAX_IGN 0}
DECL E6POS XRICK8={X 506.097260,Y -11.2192593,Z 245.251190,A -47.3005371,B -0.718434691,C 179.975281,S 2,T 3,E1 0.0,E2 0.0,E3 0.0,E4 0.0,E5 0.0,E6 0.0}
DECL FDAT Frick8={TOOL_NO 1,BASE_NO 0,IPO_FRAME #BASE,POINT2[] " ",TQ_STATE FALSE}
DECL LDAT LCPDAT59={VEL 2.00000,ACC 100.000,APO_DIST 100.000,APO_FAC 50.0000,AXIS_VEL 100.000,AXIS_ACC 100.000,ORI_TYP #VAR,CIRC_TYP #BASE,JERK_FAC 50.0000,GEAR_JERK 50.0000,EXAX_IGN 0}
DECL E6POS XIP4={X 492.207214,Y -71.4600372,Z 271.568909,A 42.5177116,B -1.73602641,C 178.891678,S 2,T 10,E1 0.0,E2 0.0,E3 0.0,E4 0.0,E5 0.0,E6 0.0}
DECL FDAT FIP4={TOOL_NO 1,BASE_NO 0,IPO_FRAME #BASE,POINT2[] " ",TQ_STATE FALSE}
DECL LDAT LCPDAT60={VEL 2.00000,ACC 100.000,APO_DIST 100.000,APO_FAC 50.0000,AXIS_VEL 100.000,AXIS_ACC 100.000,ORI_TYP #VAR,CIRC_TYP #BASE,JERK_FAC 50.0000,GEAR_JERK 50.0000,EXAX_IGN 0}
DECL E6POS Xrick9={X 494.467621,Y 75.6489792,Z 265.259155,A 45.7905807,B -3.69958639,C 177.638535,S 2,T 11,E1 0.0,E2 0.0,E3 0.0,E4 0.0,E5 0.0,E6 0.0}
DECL FDAT Frick9={TOOL_NO 1,BASE_NO 0,IPO_FRAME #BASE,POINT2[] " ",TQ_STATE FALSE}
DECL LDAT LCPDAT61={VEL 2.00000,ACC 100.000,APO_DIST 100.000,APO_FAC 50.0000,AXIS_VEL 100.000,AXIS_ACC 100.000,ORI_TYP #VAR,CIRC_TYP #BASE,JERK_FAC 50.0000,GEAR_JERK 50.0000,EXAX_IGN 0}
DECL E6POS Xrick10={X 510.444672,Y -75.1928940,Z 514.698914,A 43.6145935,B -0.547352850,C 179.277054,S 2,T 2,E1 0.0,E2 0.0,E3 0.0,E4 0.0,E5 0.0,E6 0.0}
DECL FDAT Frick10={TOOL_NO 1,BASE_NO 0,IPO_FRAME #BASE,POINT2[] " ",TQ_STATE FALSE}
DECL LDAT LCPDAT62={VEL 2.00000,ACC 100.000,APO_DIST 100.000,APO_FAC 50.0000,AXIS_VEL 100.000,AXIS_ACC 100.000,ORI_TYP #VAR,CIRC_TYP #BASE,JERK_FAC 50.0000,GEAR_JERK 50.0000,EXAX_IGN 0}
DECL E6POS Xrick11={X 510.798248,Y 70.2759705,Z 464.118958,A 44.8877525,B -0.653853238,C -179.850250,S 2,T 11,E1 0.0,E2 0.0,E3 0.0,E4 0.0,E5 0.0,E6 0.0}
DECL FDAT Frick11={TOOL_NO 1,BASE_NO 0,IPO_FRAME #BASE,POINT2[] " ",TQ_STATE FALSE}
DECL LDAT LCPDAT63={VEL 2.00000,ACC 100.000,APO_DIST 100.000,APO_FAC 50.0000,AXIS_VEL 100.000,AXIS_ACC 100.000,ORI_TYP #VAR,CIRC_TYP #BASE,JERK_FAC 50.0000,GEAR_JERK 50.0000,EXAX_IGN 0}
DECL E6POS Xrick12={X 506.097260,Y -11.2192593,Z 541.766602,A -47.3005371,B -0.718434691,C 179.975281,S 2,T 3,E1 0.0,E2 0.0,E3 0.0,E4 0.0,E5 0.0,E6 0.0}
DECL FDAT Frick12={TOOL_NO 1,BASE_NO 0,IPO_FRAME #BASE,POINT2[] " ",TQ_STATE FALSE}
DECL LDAT LCPDAT64={VEL 2.00000,ACC 100.000,APO_DIST 100.000,APO_FAC 50.0000,AXIS_VEL 100.000,AXIS_ACC 100.000,ORI_TYP #VAR,CIRC_TYP #BASE,JERK_FAC 50.0000,GEAR_JERK 50.0000,EXAX_IGN 0}
DECL LDAT LCPDAT65={VEL 2.00000,ACC 100.000,APO_DIST 100.000,APO_FAC 50.0000,AXIS_VEL 100.000,AXIS_ACC 100.000,ORI_TYP #VAR,CIRC_TYP #BASE,JERK_FAC 50.0000,GEAR_JERK 50.0000,EXAX_IGN 0}
DECL LDAT LCPDAT66={VEL 2.00000,ACC 100.000,APO_DIST 100.000,APO_FAC 50.0000,AXIS_VEL 100.000,AXIS_ACC 100.000,ORI_TYP #VAR,CIRC_TYP #BASE,JERK_FAC 50.0000,GEAR_JERK 50.0000,EXAX_IGN 0}
DECL E6POS XVENT5N={X 442.304138,Y -397.379,Z 155.349716,A -46.3701591,B 0.221998855,C 179.228592,S 2,T 2,E1 0.0,E2 0.0,E3 0.0,E4 0.0,E5 0.0,E6 0.0}
DECL FDAT Fvent5n={TOOL_NO 1,BASE_NO 0,IPO_FRAME #BASE,POINT2[] " ",TQ_STATE FALSE}
DECL LDAT LCPDAT67={VEL 2.00000,ACC 100.000,APO_DIST 100.000,APO_FAC 50.0000,AXIS_VEL 100.000,AXIS_ACC 100.000,ORI_TYP #VAR,CIRC_TYP #BASE,JERK_FAC 50.0000,GEAR_JERK 50.0000,EXAX_IGN 0}
DECL LDAT LCPDAT68={VEL 2.00000,ACC 100.000,APO_DIST 100.000,APO_FAC 50.0000,AXIS_VEL 100.000,AXIS_ACC 100.000,ORI_TYP #VAR,CIRC_TYP #BASE,JERK_FAC 50.0000,GEAR_JERK 50.0000,EXAX_IGN 0}
DECL E6POS XcodoDD5={X 146.248169,Y 296.992188,Z 337.526245,A -5.17370653,B 18.8922024,C -158.855759,S 2,T 11,E1 0.0,E2 0.0,E3 0.0,E4 0.0,E5 0.0,E6 0.0}
DECL FDAT FcodoDD5={TOOL_NO 1,BASE_NO 0,IPO_FRAME #BASE,POINT2[] " ",TQ_STATE FALSE}
DECL E6POS XVENT9AA={X 266.657104,Y -157.801224,Z 324.068085,A -140.945129,B -18.4891930,C -156.963562,S 2,T 2,E1 0.0,E2 0.0,E3 0.0,E4 0.0,E5 0.0,E6 0.0}
DECL FDAT Fvent9aa={TOOL_NO 1,BASE_NO 0,IPO_FRAME #BASE,POINT2[] " ",TQ_STATE FALSE}
DECL LDAT LCPDAT69={VEL 2.00000,ACC 100.000,APO_DIST 100.000,APO_FAC 50.0000,AXIS_VEL 100.000,AXIS_ACC 100.000,ORI_TYP #VAR,CIRC_TYP #BASE,JERK_FAC 50.0000,GEAR_JERK 50.0000,EXAX_IGN 0}
DECL E6POS XVENT10AA={X 442.283661,Y -397.354034,Z 334.883087,A -46.3715744,B 0.228786752,C 179.228363,S 2,T 2,E1 0.0,E2 0.0,E3 0.0,E4 0.0,E5 0.0,E6 0.0}
DECL FDAT Fvent10aa={TOOL_NO 1,BASE_NO 0,IPO_FRAME #BASE,POINT2[] " ",TQ_STATE FALSE}
DECL LDAT LCPDAT70={VEL 2.00000,ACC 100.000,APO_DIST 100.000,APO_FAC 50.0000,AXIS_VEL 100.000,AXIS_ACC 100.000,ORI_TYP #VAR,CIRC_TYP #BASE,JERK_FAC 50.0000,GEAR_JERK 50.0000,EXAX_IGN 0}
DECL E6POS Xrick23={X 500.839142,Y 7.79965878,Z 570.627441,A 132.153961,B 1.28462303,C -178.538376,S 2,T 35,E1 0.0,E2 0.0,E3 0.0,E4 0.0,E5 0.0,E6 0.0}
DECL FDAT Frick23={TOOL_NO 1,BASE_NO 0,IPO_FRAME #BASE,POINT2[] " ",TQ_STATE FALSE}
DECL LDAT LCPDAT99={VEL 2.00000,ACC 100.000,APO_DIST 100.000,APO_FAC 50.0000,AXIS_VEL 100.000,AXIS_ACC 100.000,ORI_TYP #VAR,CIRC_TYP #BASE,JERK_FAC 50.0000,GEAR_JERK 50.0000,EXAX_IGN 0}
DECL E6POS Xrick22={X 500.838562,Y 7.79942322,Z 241.828140,A 132.153702,B 1.28462291,C -178.538376,S 2,T 35,E1 0.0,E2 0.0,E3 0.0,E4 0.0,E5 0.0,E6 0.0}
DECL FDAT Frick22={TOOL_NO 1,BASE_NO 0,IPO_FRAME #BASE,POINT2[] " ",TQ_STATE FALSE}
DECL LDAT LCPDAT98={VEL 2.00000,ACC 100.000,APO_DIST 100.000,APO_FAC 50.0000,AXIS_VEL 100.000,AXIS_ACC 100.000,ORI_TYP #VAR,CIRC_TYP #BASE,JERK_FAC 50.0000,GEAR_JERK 50.0000,EXAX_IGN 0}
DECL E6POS Xrick21={X 500.839142,Y 7.79965878,Z 570.627441,A 132.153961,B 1.28462303,C -178.538376,S 2,T 35,E1 0.0,E2 0.0,E3 0.0,E4 0.0,E5 0.0,E6 0.0}
DECL FDAT Frick21={TOOL_NO 1,BASE_NO 0,IPO_FRAME #BASE,POINT2[] " ",TQ_STATE FALSE}
DECL LDAT LCPDAT97={VEL 2.00000,ACC 100.000,APO_DIST 100.000,APO_FAC 50.0000,AXIS_VEL 100.000,AXIS_ACC 100.000,ORI_TYP #VAR,CIRC_TYP #BASE,JERK_FAC 50.0000,GEAR_JERK 50.0000,EXAX_IGN 0}
DECL E6POS Xvent8aa_1={X 264.461761,Y 5.13799143,Z 584.457214,A 131.982437,B 1.28507471,C -178.538467,S 2,T 35,E1 0.0,E2 0.0,E3 0.0,E4 0.0,E5 0.0,E6 0.0}
DECL FDAT Fvent8aa_1={TOOL_NO 1,BASE_NO 0,IPO_FRAME #BASE,POINT2[] " ",TQ_STATE FALSE}
DECL PDAT PPDAT27={VEL 100.000,ACC 100.000,APO_DIST 100.000,APO_MODE #CDIS,GEAR_JERK 50.0000,EXAX_IGN 0}
DECL E6POS Xvent7aa_1={X 264.557251,Y -184.106232,Z 273.886200,A -139.099701,B -19.1118355,C -157.481934,S 2,T 2,E1 0.0,E2 0.0,E3 0.0,E4 0.0,E5 0.0,E6 0.0}
DECL FDAT Fvent7aa_1={TOOL_NO 1,BASE_NO 0,IPO_FRAME #BASE,POINT2[] " ",TQ_STATE FALSE}
DECL LDAT LCPDAT96={VEL 2.00000,ACC 100.000,APO_DIST 100.000,APO_FAC 50.0000,AXIS_VEL 100.000,AXIS_ACC 100.000,ORI_TYP #VAR,CIRC_TYP #BASE,JERK_FAC 50.0000,GEAR_JERK 50.0000,EXAX_IGN 0}
DECL E6POS Xvent6aa_1={X 264.557220,Y -218.268707,Z 210.296631,A -139.099686,B -19.1118259,C -157.481949,S 2,T 2,E1 0.0,E2 0.0,E3 0.0,E4 0.0,E5 0.0,E6 0.0}
DECL FDAT Fvent6aa_1={TOOL_NO 1,BASE_NO 0,IPO_FRAME #BASE,POINT2[] " ",TQ_STATE FALSE}
DECL LDAT LCPDAT95={VEL 2.00000,ACC 100.000,APO_DIST 100.000,APO_FAC 50.0000,AXIS_VEL 100.000,AXIS_ACC 100.000,ORI_TYP #VAR,CIRC_TYP #BASE,JERK_FAC 50.0000,GEAR_JERK 50.0000,EXAX_IGN 0}
DECL E6POS Xvent5n_1={X 266.034241,Y -250.412521,Z 154.373474,A -138.612717,B -20.6471786,C -158.911987,S 2,T 2,E1 0.0,E2 0.0,E3 0.0,E4 0.0,E5 0.0,E6 0.0}
DECL FDAT Fvent5n_1={TOOL_NO 1,BASE_NO 0,IPO_FRAME #BASE,POINT2[] " ",TQ_STATE FALSE}
DECL LDAT LCPDAT94={VEL 2.00000,ACC 100.000,APO_DIST 100.000,APO_FAC 50.0000,AXIS_VEL 100.000,AXIS_ACC 100.000,ORI_TYP #VAR,CIRC_TYP #BASE,JERK_FAC 50.0000,GEAR_JERK 50.0000,EXAX_IGN 0}
DECL E6POS Xvent10aa_1={X 266.973511,Y -220.491226,Z 198.112228,A -138.612717,B -20.6471786,C -158.911987,S 2,T 2,E1 0.0,E2 0.0,E3 0.0,E4 0.0,E5 0.0,E6 0.0}
DECL FDAT Fvent10aa_1={TOOL_NO 1,BASE_NO 0,IPO_FRAME #BASE,POINT2[] " ",TQ_STATE FALSE}
DECL LDAT LCPDAT93={VEL 2.00000,ACC 100.000,APO_DIST 100.000,APO_FAC 50.0000,AXIS_VEL 100.000,AXIS_ACC 100.000,ORI_TYP #VAR,CIRC_TYP #BASE,JERK_FAC 50.0000,GEAR_JERK 50.0000,EXAX_IGN 0}
DECL E6POS Xvent4aa_1={X 264.553955,Y -220.491226,Z 198.112228,A -139.098389,B -19.1098919,C -157.483841,S 2,T 2,E1 0.0,E2 0.0,E3 0.0,E4 0.0,E5 0.0,E6 0.0}
DECL FDAT Fvent4aa_1={TOOL_NO 1,BASE_NO 0,IPO_FRAME #BASE,POINT2[] " ",TQ_STATE FALSE}
DECL LDAT LCPDAT92={VEL 2.00000,ACC 100.000,APO_DIST 100.000,APO_FAC 50.0000,AXIS_VEL 100.000,AXIS_ACC 100.000,ORI_TYP #VAR,CIRC_TYP #BASE,JERK_FAC 50.0000,GEAR_JERK 50.0000,EXAX_IGN 0}
DECL E6POS Xvent3aa_1={X 264.549,Y -226.508316,Z 557.449402,A -139.096802,B -19.1079426,C -157.486145,S 2,T 2,E1 0.0,E2 0.0,E3 0.0,E4 0.0,E5 0.0,E6 0.0}
DECL FDAT Fvent3aa_1={TOOL_NO 1,BASE_NO 0,IPO_FRAME #BASE,POINT2[] " ",TQ_STATE FALSE}
DECL PDAT PPDAT26={VEL 100.000,ACC 100.000,APO_DIST 100.000,APO_MODE #CDIS,GEAR_JERK 50.0000,EXAX_IGN 0}
DECL E6POS XventA4={X 415.256256,Y -14.7377806,Z 509.505,A -46.3701591,B 0.221998855,C 179.228592,S 2,T 2,E1 0.0,E2 0.0,E3 0.0,E4 0.0,E5 0.0,E6 0.0}
DECL FDAT FventA4={TOOL_NO 1,BASE_NO 0,IPO_FRAME #BASE,POINT2[] " ",TQ_STATE FALSE}
DECL PDAT PPDAT25={VEL 100.000,ACC 100.000,APO_DIST 100.000,APO_MODE #CDIS,GEAR_JERK 50.0000,EXAX_IGN 0}
DECL E6POS Xrick20={X 518.938049,Y 70.2749329,Z 506.411896,A 44.8877525,B -0.653846,C -179.850266,S 2,T 11,E1 0.0,E2 0.0,E3 0.0,E4 0.0,E5 0.0,E6 0.0}
DECL FDAT Frick20={TOOL_NO 1,BASE_NO 0,IPO_FRAME #BASE,POINT2[] " ",TQ_STATE FALSE}
DECL LDAT LCPDAT91={VEL 2.00000,ACC 100.000,APO_DIST 100.000,APO_FAC 50.0000,AXIS_VEL 100.000,AXIS_ACC 100.000,ORI_TYP #VAR,CIRC_TYP #BASE,JERK_FAC 50.0000,GEAR_JERK 50.0000,EXAX_IGN 0}
DECL E6POS Xrick19={X 518.938049,Y 70.2749329,Z 342.100342,A 44.8877525,B -0.653846,C -179.850266,S 2,T 11,E1 0.0,E2 0.0,E3 0.0,E4 0.0,E5 0.0,E6 0.0}
DECL FDAT Frick19={TOOL_NO 1,BASE_NO 0,IPO_FRAME #BASE,POINT2[] " ",TQ_STATE FALSE}
DECL LDAT LCPDAT90={VEL 2.00000,ACC 100.000,APO_DIST 100.000,APO_FAC 50.0000,AXIS_VEL 100.000,AXIS_ACC 100.000,ORI_TYP #VAR,CIRC_TYP #BASE,JERK_FAC 50.0000,GEAR_JERK 50.0000,EXAX_IGN 0}
DECL E6POS Xrick18={X 518.938049,Y 70.2749329,Z 506.411896,A 44.8877525,B -0.653846,C -179.850266,S 2,T 11,E1 0.0,E2 0.0,E3 0.0,E4 0.0,E5 0.0,E6 0.0}
DECL FDAT Frick18={TOOL_NO 1,BASE_NO 0,IPO_FRAME #BASE,POINT2[] " ",TQ_STATE FALSE}
DECL LDAT LCPDAT89={VEL 2.00000,ACC 100.000,APO_DIST 100.000,APO_FAC 50.0000,AXIS_VEL 100.000,AXIS_ACC 100.000,ORI_TYP #VAR,CIRC_TYP #BASE,JERK_FAC 50.0000,GEAR_JERK 50.0000,EXAX_IGN 0}
DECL E6POS XPD_2={X 496.200287,Y 374.316742,Z 330.279724,A 43.3064499,B -1.60716689,C 179.054642,S 2,T 3,E1 0.0,E2 0.0,E3 0.0,E4 0.0,E5 0.0,E6 0.0}
DECL FDAT FPD_2={TOOL_NO 1,BASE_NO 0,IPO_FRAME #BASE,POINT2[] " ",TQ_STATE FALSE}
DECL LDAT LCPDAT88={VEL 2.00000,ACC 100.000,APO_DIST 100.000,APO_FAC 50.0000,AXIS_VEL 100.000,AXIS_ACC 100.000,ORI_TYP #VAR,CIRC_TYP #BASE,JERK_FAC 50.0000,GEAR_JERK 50.0000,EXAX_IGN 0}
DECL E6POS XPDA_2={X 496.200287,Y 374.316742,Z 450.351959,A 43.3064499,B -1.60716689,C 179.054642,S 2,T 3,E1 0.0,E2 0.0,E3 0.0,E4 0.0,E5 0.0,E6 0.0}
DECL FDAT FPDA_2={TOOL_NO 1,BASE_NO 0,IPO_FRAME #BASE,POINT2[] " ",TQ_STATE FALSE}
DECL LDAT LCPDAT87={VEL 2.00000,ACC 100.000,APO_DIST 100.000,APO_FAC 50.0000,AXIS_VEL 100.000,AXIS_ACC 100.000,ORI_TYP #VAR,CIRC_TYP #BASE,JERK_FAC 50.0000,GEAR_JERK 50.0000,EXAX_IGN 0}
DECL E6POS Xrick17={X 500.487122,Y -75.3265762,Z 470.598694,A 42.9319191,B -1.89823210,C 177.983963,S 2,T 10,E1 0.0,E2 0.0,E3 0.0,E4 0.0,E5 0.0,E6 0.0}
DECL FDAT Frick17={TOOL_NO 1,BASE_NO 0,IPO_FRAME #BASE,POINT2[] " ",TQ_STATE FALSE}
DECL LDAT LCPDAT86={VEL 2.00000,ACC 100.000,APO_DIST 100.000,APO_FAC 50.0000,AXIS_VEL 100.000,AXIS_ACC 100.000,ORI_TYP #VAR,CIRC_TYP #BASE,JERK_FAC 50.0000,GEAR_JERK 50.0000,EXAX_IGN 0}
DECL E6POS Xrick16={X 500.487122,Y -75.3265762,Z 341.885,A 42.9319191,B -1.89823210,C 177.983963,S 2,T 42,E1 0.0,E2 0.0,E3 0.0,E4 0.0,E5 0.0,E6 0.0}
DECL FDAT Frick16={TOOL_NO 1,BASE_NO 0,IPO_FRAME #BASE,POINT2[] " ",TQ_STATE FALSE}
DECL LDAT LCPDAT85={VEL 2.00000,ACC 100.000,APO_DIST 100.000,APO_FAC 50.0000,AXIS_VEL 100.000,AXIS_ACC 100.000,ORI_TYP #VAR,CIRC_TYP #BASE,JERK_FAC 50.0000,GEAR_JERK 50.0000,EXAX_IGN 0}
DECL E6POS Xrick15={X 500.487122,Y -75.3265762,Z 470.598694,A 42.9319191,B -1.89823210,C 177.983963,S 2,T 10,E1 0.0,E2 0.0,E3 0.0,E4 0.0,E5 0.0,E6 0.0}
DECL FDAT Frick15={TOOL_NO 1,BASE_NO 0,IPO_FRAME #BASE,POINT2[] " ",TQ_STATE FALSE}
DECL LDAT LCPDAT84={VEL 2.00000,ACC 100.000,APO_DIST 100.000,APO_FAC 50.0000,AXIS_VEL 100.000,AXIS_ACC 100.000,ORI_TYP #VAR,CIRC_TYP #BASE,JERK_FAC 50.0000,GEAR_JERK 50.0000,EXAX_IGN 0}
DECL E6POS XPI_2={X 488.794952,Y 263.522217,Z 330.558746,A 38.9071503,B -1.58586621,C 179.083191,S 2,T 3,E1 0.0,E2 0.0,E3 0.0,E4 0.0,E5 0.0,E6 0.0}
DECL FDAT FPI_2={TOOL_NO 1,BASE_NO 0,IPO_FRAME #BASE,POINT2[] " ",TQ_STATE FALSE}
DECL LDAT LCPDAT83={VEL 2.00000,ACC 100.000,APO_DIST 100.000,APO_FAC 50.0000,AXIS_VEL 100.000,AXIS_ACC 100.000,ORI_TYP #VAR,CIRC_TYP #BASE,JERK_FAC 50.0000,GEAR_JERK 50.0000,EXAX_IGN 0}
DECL E6POS XPIA_2={X 488.794952,Y 263.522217,Z 467.844391,A 38.9071503,B -1.58586633,C 179.083191,S 2,T 3,E1 0.0,E2 0.0,E3 0.0,E4 0.0,E5 0.0,E6 0.0}
DECL FDAT FPIA_2={TOOL_NO 1,BASE_NO 0,IPO_FRAME #BASE,POINT2[] " ",TQ_STATE FALSE}
DECL LDAT LCPDAT82={VEL 2.00000,ACC 100.000,APO_DIST 100.000,APO_FAC 50.0000,AXIS_VEL 100.000,AXIS_ACC 100.000,ORI_TYP #VAR,CIRC_TYP #BASE,JERK_FAC 50.0000,GEAR_JERK 50.0000,EXAX_IGN 0}
DECL E6POS Xrick14={X 494.467621,Y 75.6489792,Z 265.259155,A 45.7905807,B -3.69958639,C 177.638535,S 2,T 11,E1 0.0,E2 0.0,E3 0.0,E4 0.0,E5 0.0,E6 0.0}
DECL FDAT Frick14={TOOL_NO 1,BASE_NO 0,IPO_FRAME #BASE,POINT2[] " ",TQ_STATE FALSE}
DECL LDAT LCPDAT81={VEL 2.00000,ACC 100.000,APO_DIST 100.000,APO_FAC 50.0000,AXIS_VEL 100.000,AXIS_ACC 100.000,ORI_TYP #VAR,CIRC_TYP #BASE,JERK_FAC 50.0000,GEAR_JERK 50.0000,EXAX_IGN 0}
DECL E6POS Xrick_1={X 494.508514,Y 75.6534,Z 119.691635,A 45.7914047,B -3.70587182,C 177.634262,S 2,T 11,E1 0.0,E2 0.0,E3 0.0,E4 0.0,E5 0.0,E6 0.0}
DECL FDAT Frick_1={TOOL_NO 1,BASE_NO 0,IPO_FRAME #BASE,POINT2[] " ",TQ_STATE FALSE}
DECL LDAT LCPDAT80={VEL 2.00000,ACC 100.000,APO_DIST 100.000,APO_FAC 50.0000,AXIS_VEL 100.000,AXIS_ACC 100.000,ORI_TYP #VAR,CIRC_TYP #BASE,JERK_FAC 50.0000,GEAR_JERK 50.0000,EXAX_IGN 0}
DECL E6POS Xrick13={X 494.467621,Y 75.6489792,Z 265.259155,A 45.7905807,B -3.69958639,C 177.638535,S 2,T 11,E1 0.0,E2 0.0,E3 0.0,E4 0.0,E5 0.0,E6 0.0}
DECL FDAT Frick13={TOOL_NO 1,BASE_NO 0,IPO_FRAME #BASE,POINT2[] " ",TQ_STATE FALSE}
DECL LDAT LCPDAT79={VEL 2.00000,ACC 100.000,APO_DIST 100.000,APO_FAC 50.0000,AXIS_VEL 100.000,AXIS_ACC 100.000,ORI_TYP #VAR,CIRC_TYP #BASE,JERK_FAC 50.0000,GEAR_JERK 50.0000,EXAX_IGN 0}
DECL E6POS Xcentro_5_1={X 222.017685,Y 1.93147576,Z 503.686340,A 38.9071503,B -1.58586597,C 179.083191,S 2,T 10,E1 0.0,E2 0.0,E3 0.0,E4 0.0,E5 0.0,E6 0.0}
DECL FDAT Fcentro_5_1={TOOL_NO 1,BASE_NO 0,IPO_FRAME #BASE,POINT2[] " ",TQ_STATE FALSE}
DECL PDAT PPDAT24={VEL 100.000,ACC 100.000,APO_DIST 100.000,APO_MODE #CDIS,GEAR_JERK 50.0000,EXAX_IGN 0}
DECL E6POS XcodoDD6={X 146.248169,Y 296.992188,Z 337.526245,A -5.17370653,B 18.8922024,C -158.855759,S 2,T 11,E1 0.0,E2 0.0,E3 0.0,E4 0.0,E5 0.0,E6 0.0}
DECL FDAT FcodoDD6={TOOL_NO 1,BASE_NO 0,IPO_FRAME #BASE,POINT2[] " ",TQ_STATE FALSE}
DECL LDAT LCPDAT78={VEL 2.00000,ACC 100.000,APO_DIST 100.000,APO_FAC 50.0000,AXIS_VEL 100.000,AXIS_ACC 100.000,ORI_TYP #VAR,CIRC_TYP #BASE,JERK_FAC 50.0000,GEAR_JERK 50.0000,EXAX_IGN 0}
DECL E6POS XcodoD8={X 124.531929,Y 329.923431,Z 264.745789,A -5.13479567,B 18.8223400,C -158.743607,S 2,T 11,E1 0.0,E2 0.0,E3 0.0,E4 0.0,E5 0.0,E6 0.0}
DECL FDAT FcodoD8={TOOL_NO 1,BASE_NO 0,IPO_FRAME #BASE,POINT2[] " ",TQ_STATE FALSE}
DECL LDAT LCPDAT77={VEL 2.00000,ACC 100.000,APO_DIST 100.000,APO_FAC 50.0000,AXIS_VEL 100.000,AXIS_ACC 100.000,ORI_TYP #VAR,CIRC_TYP #BASE,JERK_FAC 50.0000,GEAR_JERK 50.0000,EXAX_IGN 0}
DECL E6POS XcodoD7={X 120.584869,Y 330.035919,Z 422.057,A -5.40004730,B 17.7066059,C -156.192,S 2,T 11,E1 0.0,E2 0.0,E3 0.0,E4 0.0,E5 0.0,E6 0.0}
DECL FDAT FcodoD7={TOOL_NO 1,BASE_NO 0,IPO_FRAME #BASE,POINT2[] " ",TQ_STATE FALSE}
DECL PDAT PPDAT23={VEL 100.000,ACC 100.000,APO_DIST 100.000,APO_MODE #CDIS,GEAR_JERK 50.0000,EXAX_IGN 0}
DECL E6POS XIP7={X 492.207214,Y -71.4600372,Z 271.568909,A 42.5177116,B -1.73602641,C 178.891678,S 2,T 10,E1 0.0,E2 0.0,E3 0.0,E4 0.0,E5 0.0,E6 0.0}
DECL FDAT FIP7={TOOL_NO 1,BASE_NO 0,IPO_FRAME #BASE,POINT2[] " ",TQ_STATE FALSE}
DECL LDAT LCPDAT76={VEL 2.00000,ACC 100.000,APO_DIST 100.000,APO_FAC 50.0000,AXIS_VEL 100.000,AXIS_ACC 100.000,ORI_TYP #VAR,CIRC_TYP #BASE,JERK_FAC 50.0000,GEAR_JERK 50.0000,EXAX_IGN 0}
DECL E6POS XIP6={X 493.945343,Y -71.5176544,Z 120.988960,A 42.5177116,B -1.73602641,C 178.891678,S 2,T 10,E1 0.0,E2 0.0,E3 0.0,E4 0.0,E5 0.0,E6 0.0}
DECL FDAT FIP6={TOOL_NO 1,BASE_NO 0,IPO_FRAME #BASE,POINT2[] " ",TQ_STATE FALSE}
DECL LDAT LCPDAT75={VEL 2.00000,ACC 100.000,APO_DIST 100.000,APO_FAC 50.0000,AXIS_VEL 100.000,AXIS_ACC 100.000,ORI_TYP #VAR,CIRC_TYP #BASE,JERK_FAC 50.0000,GEAR_JERK 50.0000,EXAX_IGN 0}
DECL E6POS XIP5={X 492.207214,Y -71.4600372,Z 271.568909,A 42.5177116,B -1.73602641,C 178.891678,S 2,T 10,E1 0.0,E2 0.0,E3 0.0,E4 0.0,E5 0.0,E6 0.0}
DECL FDAT FIP5={TOOL_NO 1,BASE_NO 0,IPO_FRAME #BASE,POINT2[] " ",TQ_STATE FALSE}
DECL LDAT LCPDAT74={VEL 2.00000,ACC 100.000,APO_DIST 100.000,APO_FAC 50.0000,AXIS_VEL 100.000,AXIS_ACC 100.000,ORI_TYP #VAR,CIRC_TYP #BASE,JERK_FAC 50.0000,GEAR_JERK 50.0000,EXAX_IGN 0}
DECL E6POS XIB4={X 172.239731,Y 269.638824,Z 111.731445,A -6.09838581,B 20.0551949,C -158.106277,S 2,T 11,E1 0.0,E2 0.0,E3 0.0,E4 0.0,E5 0.0,E6 0.0}
DECL FDAT FIB4={TOOL_NO 1,BASE_NO 0,IPO_FRAME #BASE,POINT2[] " ",TQ_STATE FALSE}
DECL LDAT LCPDAT73={VEL 2.00000,ACC 100.000,APO_DIST 100.000,APO_FAC 50.0000,AXIS_VEL 100.000,AXIS_ACC 100.000,ORI_TYP #VAR,CIRC_TYP #BASE,JERK_FAC 50.0000,GEAR_JERK 50.0000,EXAX_IGN 0}
DECL E6POS XcodoIB7={X 169.370163,Y 288.233887,Z 215.088318,A -9.98564243,B -1.58595812,C 179.083130,S 2,T 3,E1 0.0,E2 0.0,E3 0.0,E4 0.0,E5 0.0,E6 0.0}
DECL FDAT FcodoIB7={TOOL_NO 1,BASE_NO 0,IPO_FRAME #BASE,POINT2[] " ",TQ_STATE FALSE}
DECL LDAT LCPDAT72={VEL 2.00000,ACC 100.000,APO_DIST 100.000,APO_FAC 50.0000,AXIS_VEL 100.000,AXIS_ACC 100.000,ORI_TYP #VAR,CIRC_TYP #BASE,JERK_FAC 50.0000,GEAR_JERK 50.0000,EXAX_IGN 0}
DECL E6POS XcodoIB6={X 169.372009,Y 288.237305,Z 503.685242,A -9.98564529,B -1.58597386,C 179.083130,S 2,T 3,E1 0.0,E2 0.0,E3 0.0,E4 0.0,E5 0.0,E6 0.0}
DECL FDAT FcodoIB6={TOOL_NO 1,BASE_NO 0,IPO_FRAME #BASE,POINT2[] " ",TQ_STATE FALSE}
DECL LDAT LCPDAT71={VEL 2.00000,ACC 100.000,APO_DIST 100.000,APO_FAC 50.0000,AXIS_VEL 100.000,AXIS_ACC 100.000,ORI_TYP #VAR,CIRC_TYP #BASE,JERK_FAC 50.0000,GEAR_JERK 50.0000,EXAX_IGN 0}
DECL E6POS Xcentro_6={X 222.017685,Y 1.93147576,Z 503.686340,A 38.9071503,B -1.58586597,C 179.083191,S 2,T 10,E1 0.0,E2 0.0,E3 0.0,E4 0.0,E5 0.0,E6 0.0}
DECL FDAT Fcentro_6={TOOL_NO 1,BASE_NO 0,IPO_FRAME #BASE,POINT2[] " ",TQ_STATE FALSE}
DECL PDAT PPDAT22={VEL 100.000,ACC 100.000,APO_DIST 100.000,APO_MODE #CDIS,GEAR_JERK 50.0000,EXAX_IGN 0}
DECL E6POS XFRED2PI22={X 441.488434,Y 263.522217,Z 330.558746,A 38.9071503,B -1.58586657,C 179.083191,S 2,T 3,E1 0.0,E2 0.0,E3 0.0,E4 0.0,E5 0.0,E6 0.0}
DECL FDAT Ffred2PI22={TOOL_NO 1,BASE_NO 0,IPO_FRAME #BASE,POINT2[] " ",TQ_STATE FALSE}
DECL LDAT LCPDAT100={VEL 2.00000,ACC 100.000,APO_DIST 100.000,APO_FAC 50.0000,AXIS_VEL 100.000,AXIS_ACC 100.000,ORI_TYP #VAR,CIRC_TYP #BASE,JERK_FAC 50.0000,GEAR_JERK 50.0000,EXAX_IGN 0}
DECL E6POS XFRED2PI23={X 441.300446,Y 263.400269,Z 471.415405,A 38.9080505,B -1.52164364,C 179.091858,S 2,T 3,E1 0.0,E2 0.0,E3 0.0,E4 0.0,E5 0.0,E6 0.0}
DECL FDAT Ffred2PI23={TOOL_NO 1,BASE_NO 0,IPO_FRAME #BASE,POINT2[] " ",TQ_STATE FALSE}
DECL LDAT LCPDAT101={VEL 2.00000,ACC 100.000,APO_DIST 100.000,APO_FAC 50.0000,AXIS_VEL 100.000,AXIS_ACC 100.000,ORI_TYP #VAR,CIRC_TYP #BASE,JERK_FAC 50.0000,GEAR_JERK 50.0000,EXAX_IGN 0}
DECL E6POS Xfred2PI24={X 441.300446,Y 263.400269,Z 471.415405,A 38.9080505,B -1.52164364,C 179.091858,S 2,T 3,E1 0.0,E2 0.0,E3 0.0,E4 0.0,E5 0.0,E6 0.0}
DECL FDAT Ffred2PI24={TOOL_NO 1,BASE_NO 0,IPO_FRAME #BASE,POINT2[] " ",TQ_STATE FALSE}
DECL LDAT LCPDAT102={VEL 2.00000,ACC 100.000,APO_DIST 100.000,APO_FAC 50.0000,AXIS_VEL 100.000,AXIS_ACC 100.000,ORI_TYP #VAR,CIRC_TYP #BASE,JERK_FAC 50.0000,GEAR_JERK 50.0000,EXAX_IGN 0}
DECL E6POS XFRED2PD2={X 445.212769,Y 374.316742,Z 330.279724,A 43.3064499,B -1.60716689,C 179.054642,S 2,T 3,E1 0.0,E2 0.0,E3 0.0,E4 0.0,E5 0.0,E6 0.0}
DECL FDAT Ffred2PD2={TOOL_NO 1,BASE_NO 0,IPO_FRAME #BASE,POINT2[] " ",TQ_STATE FALSE}
DECL LDAT LCPDAT103={VEL 2.00000,ACC 100.000,APO_DIST 100.000,APO_FAC 50.0000,AXIS_VEL 100.000,AXIS_ACC 100.000,ORI_TYP #VAR,CIRC_TYP #BASE,JERK_FAC 50.0000,GEAR_JERK 50.0000,EXAX_IGN 0}
DECL E6POS XFRED2PDA3={X 445.212769,Y 374.316742,Z 452.541840,A 43.3064499,B -1.60716701,C 179.054642,S 2,T 3,E1 0.0,E2 0.0,E3 0.0,E4 0.0,E5 0.0,E6 0.0}
DECL FDAT Ffred2PDA3={TOOL_NO 1,BASE_NO 0,IPO_FRAME #BASE,POINT2[] " ",TQ_STATE FALSE}
DECL LDAT LCPDAT104={VEL 2.00000,ACC 100.000,APO_DIST 100.000,APO_FAC 50.0000,AXIS_VEL 100.000,AXIS_ACC 100.000,ORI_TYP #VAR,CIRC_TYP #BASE,JERK_FAC 50.0000,GEAR_JERK 50.0000,EXAX_IGN 0}
DECL E6POS Xfred2PDA4={X 445.212769,Y 374.316742,Z 452.541840,A 43.3064499,B -1.60716701,C 179.054642,S 2,T 3,E1 0.0,E2 0.0,E3 0.0,E4 0.0,E5 0.0,E6 0.0}
DECL FDAT Ffred2PDA4={TOOL_NO 1,BASE_NO 0,IPO_FRAME #BASE,POINT2[] " ",TQ_STATE FALSE}
DECL LDAT LCPDAT105={VEL 2.00000,ACC 100.000,APO_DIST 100.000,APO_FAC 50.0000,AXIS_VEL 100.000,AXIS_ACC 100.000,ORI_TYP #VAR,CIRC_TYP #BASE,JERK_FAC 50.0000,GEAR_JERK 50.0000,EXAX_IGN 0}
DECL E6POS Xrick34={X 500.839142,Y 7.79965878,Z 570.627441,A 132.153961,B 1.28462303,C -178.538376,S 2,T 35,E1 0.0,E2 0.0,E3 0.0,E4 0.0,E5 0.0,E6 0.0}
DECL FDAT Frick34={TOOL_NO 1,BASE_NO 0,IPO_FRAME #BASE,POINT2[] " ",TQ_STATE FALSE}
DECL LDAT LCPDAT134={VEL 2.00000,ACC 100.000,APO_DIST 100.000,APO_FAC 50.0000,AXIS_VEL 100.000,AXIS_ACC 100.000,ORI_TYP #VAR,CIRC_TYP #BASE,JERK_FAC 50.0000,GEAR_JERK 50.0000,EXAX_IGN 0}
DECL E6POS Xrick33={X 500.838562,Y 7.79942322,Z 241.828140,A 132.153702,B 1.28462291,C -178.538376,S 2,T 35,E1 0.0,E2 0.0,E3 0.0,E4 0.0,E5 0.0,E6 0.0}
DECL FDAT Frick33={TOOL_NO 1,BASE_NO 0,IPO_FRAME #BASE,POINT2[] " ",TQ_STATE FALSE}
DECL LDAT LCPDAT133={VEL 2.00000,ACC 100.000,APO_DIST 100.000,APO_FAC 50.0000,AXIS_VEL 100.000,AXIS_ACC 100.000,ORI_TYP #VAR,CIRC_TYP #BASE,JERK_FAC 50.0000,GEAR_JERK 50.0000,EXAX_IGN 0}
DECL E6POS Xrick32={X 500.839142,Y 7.79965878,Z 570.627441,A 132.153961,B 1.28462303,C -178.538376,S 2,T 35,E1 0.0,E2 0.0,E3 0.0,E4 0.0,E5 0.0,E6 0.0}
DECL FDAT Frick32={TOOL_NO 1,BASE_NO 0,IPO_FRAME #BASE,POINT2[] " ",TQ_STATE FALSE}
DECL LDAT LCPDAT132={VEL 2.00000,ACC 100.000,APO_DIST 100.000,APO_FAC 50.0000,AXIS_VEL 100.000,AXIS_ACC 100.000,ORI_TYP #VAR,CIRC_TYP #BASE,JERK_FAC 50.0000,GEAR_JERK 50.0000,EXAX_IGN 0}
DECL E6POS Xvent8aa_2={X 264.461761,Y 5.13799143,Z 584.457214,A 131.982437,B 1.28507471,C -178.538467,S 2,T 35,E1 0.0,E2 0.0,E3 0.0,E4 0.0,E5 0.0,E6 0.0}
DECL FDAT Fvent8aa_2={TOOL_NO 1,BASE_NO 0,IPO_FRAME #BASE,POINT2[] " ",TQ_STATE FALSE}
DECL PDAT PPDAT33={VEL 100.000,ACC 100.000,APO_DIST 100.000,APO_MODE #CDIS,GEAR_JERK 50.0000,EXAX_IGN 0}
DECL E6POS Xvent7aa_2={X 264.557251,Y -184.106232,Z 273.886200,A -139.099701,B -19.1118355,C -157.481934,S 2,T 2,E1 0.0,E2 0.0,E3 0.0,E4 0.0,E5 0.0,E6 0.0}
DECL FDAT Fvent7aa_2={TOOL_NO 1,BASE_NO 0,IPO_FRAME #BASE,POINT2[] " ",TQ_STATE FALSE}
DECL LDAT LCPDAT131={VEL 2.00000,ACC 100.000,APO_DIST 100.000,APO_FAC 50.0000,AXIS_VEL 100.000,AXIS_ACC 100.000,ORI_TYP #VAR,CIRC_TYP #BASE,JERK_FAC 50.0000,GEAR_JERK 50.0000,EXAX_IGN 0}
DECL E6POS Xvent6aa_2={X 264.557220,Y -218.268707,Z 210.296631,A -139.099686,B -19.1118259,C -157.481949,S 2,T 2,E1 0.0,E2 0.0,E3 0.0,E4 0.0,E5 0.0,E6 0.0}
DECL FDAT Fvent6aa_2={TOOL_NO 1,BASE_NO 0,IPO_FRAME #BASE,POINT2[] " ",TQ_STATE FALSE}
DECL LDAT LCPDAT130={VEL 2.00000,ACC 100.000,APO_DIST 100.000,APO_FAC 50.0000,AXIS_VEL 100.000,AXIS_ACC 100.000,ORI_TYP #VAR,CIRC_TYP #BASE,JERK_FAC 50.0000,GEAR_JERK 50.0000,EXAX_IGN 0}
DECL E6POS Xvent5n_2={X 266.034241,Y -250.412521,Z 154.373474,A -138.612717,B -20.6471786,C -158.911987,S 2,T 2,E1 0.0,E2 0.0,E3 0.0,E4 0.0,E5 0.0,E6 0.0}
DECL FDAT Fvent5n_2={TOOL_NO 1,BASE_NO 0,IPO_FRAME #BASE,POINT2[] " ",TQ_STATE FALSE}
DECL LDAT LCPDAT129={VEL 2.00000,ACC 100.000,APO_DIST 100.000,APO_FAC 50.0000,AXIS_VEL 100.000,AXIS_ACC 100.000,ORI_TYP #VAR,CIRC_TYP #BASE,JERK_FAC 50.0000,GEAR_JERK 50.0000,EXAX_IGN 0}
DECL E6POS Xvent10aa_2={X 266.973511,Y -220.491226,Z 198.112228,A -138.612717,B -20.6471786,C -158.911987,S 2,T 2,E1 0.0,E2 0.0,E3 0.0,E4 0.0,E5 0.0,E6 0.0}
DECL FDAT Fvent10aa_2={TOOL_NO 1,BASE_NO 0,IPO_FRAME #BASE,POINT2[] " ",TQ_STATE FALSE}
DECL LDAT LCPDAT128={VEL 2.00000,ACC 100.000,APO_DIST 100.000,APO_FAC 50.0000,AXIS_VEL 100.000,AXIS_ACC 100.000,ORI_TYP #VAR,CIRC_TYP #BASE,JERK_FAC 50.0000,GEAR_JERK 50.0000,EXAX_IGN 0}
DECL E6POS Xvent4aa_2={X 264.553955,Y -220.491226,Z 198.112228,A -139.098389,B -19.1098919,C -157.483841,S 2,T 2,E1 0.0,E2 0.0,E3 0.0,E4 0.0,E5 0.0,E6 0.0}
DECL FDAT Fvent4aa_2={TOOL_NO 1,BASE_NO 0,IPO_FRAME #BASE,POINT2[] " ",TQ_STATE FALSE}
DECL LDAT LCPDAT127={VEL 2.00000,ACC 100.000,APO_DIST 100.000,APO_FAC 50.0000,AXIS_VEL 100.000,AXIS_ACC 100.000,ORI_TYP #VAR,CIRC_TYP #BASE,JERK_FAC 50.0000,GEAR_JERK 50.0000,EXAX_IGN 0}
DECL E6POS Xvent3aa_2={X 264.549,Y -226.508316,Z 557.449402,A -139.096802,B -19.1079426,C -157.486145,S 2,T 2,E1 0.0,E2 0.0,E3 0.0,E4 0.0,E5 0.0,E6 0.0}
DECL FDAT Fvent3aa_2={TOOL_NO 1,BASE_NO 0,IPO_FRAME #BASE,POINT2[] " ",TQ_STATE FALSE}
DECL PDAT PPDAT32={VEL 100.000,ACC 100.000,APO_DIST 100.000,APO_MODE #CDIS,GEAR_JERK 50.0000,EXAX_IGN 0}
DECL E6POS XventA5={X 415.256256,Y -14.7377806,Z 509.505,A -46.3701591,B 0.221998855,C 179.228592,S 2,T 2,E1 0.0,E2 0.0,E3 0.0,E4 0.0,E5 0.0,E6 0.0}
DECL FDAT FventA5={TOOL_NO 1,BASE_NO 0,IPO_FRAME #BASE,POINT2[] " ",TQ_STATE FALSE}
DECL PDAT PPDAT31={VEL 100.000,ACC 100.000,APO_DIST 100.000,APO_MODE #CDIS,GEAR_JERK 50.0000,EXAX_IGN 0}
DECL E6POS Xrick31={X 518.938049,Y 70.2749329,Z 506.411896,A 44.8877525,B -0.653846,C -179.850266,S 2,T 11,E1 0.0,E2 0.0,E3 0.0,E4 0.0,E5 0.0,E6 0.0}
DECL FDAT Frick31={TOOL_NO 1,BASE_NO 0,IPO_FRAME #BASE,POINT2[] " ",TQ_STATE FALSE}
